      NOP   0;
// CO2D6RV1 PID 001 CO2 D6 RV1
      CALL FC    55 (
           UnitNo                   := #UnitNo,
           PIDRec                   := DB2346.CO2D6RV1,
           SpExt                    := DB2346.DBD  234,
           PVal                     := DB2346.DBD  254,
           OPer                     := PQW  544);

NETWORK
TITLE =unit supply

      UC    FB [#UnitFB];

NETWORK
TITLE =D6_G1  D6_G1
// Act 001
// Box           : VS2-BB
// Output address: Q310.2
      CALL FC    70 (
           UnitNo                   := #UnitNo,
           ActRec                   := DB2340.D6_G1,
           Typ                      := 1,
           FBa                      := #xTmp,
           FBa2                     := I    310.2,
           Out                      := Q    310.2);

NETWORK
TITLE =CO2_D6V2  Ansteuerung D6V2
// Act 002
// Box           : CO2 Dosierung
// Output address: Q61.4
      CALL FC    70 (
           UnitNo                   := #UnitNo,
           ActRec                   := DB2340.CO2_D6V2,
           Typ                      := 0,
           FBa                      := #xTmp,
           FBa2                     := #xTmp,
           Out                      := Q     61.4);

NETWORK
TITLE =CO2_D6V1  Ansteuerung D6V1
// Act 003
// Box           : CO2 Dosierung
// Output address: Q60.4
      CALL FC    70 (
           UnitNo                   := #UnitNo,
           ActRec                   := DB2340.CO2_D6V1,
           Typ                      := 0,
           FBa                      := #xTmp,
           FBa2                     := #xTmp,
           Out                      := Q     60.4);

NETWORK
TITLE =D6RV1  CO2 D6 RV1
// Act 004
// Box           :
// Input address : #xtmp
// Output address: #xtmp
      CALL FC    70 (
           UnitNo                   := #UnitNo,
           ActRec                   := DB2340.D6RV1,
           Typ                      := 4,
           FBa                      := #xTmp,
           FBa2                     := #xTmp,
           Out                      := #xTmp);

END_FUNCTION_BLOCK

FUNCTION_BLOCK FB 1341
TITLE =U034: Well Transfer D6
FAMILY : BOTEC_F1
NAME : UniE
VERSION : 1.2


VAR_TEMP
  CIP : BOOL ;	//CIP active
  UNIM : BOOL ;	//Unit Not In Maintenance
  GenRel : BOOL ;	//general OK (emergency and maintenance OK)
  EStopOK : BOOL ;	//emergency OK
  UnitNo : INT ;	//unit number
  xTmp : BOOL ;	//Temporary Bool
  iTmp : INT ;	//Temporary INT
  rTmp : REAL ;	//Temporary REAL
  dTmp : DINT ;	//Temporary DINT (free for general use)
  RetValInt : INT ;	//return value
END_VAR
BEGIN
NETWORK
TITLE =General

      SET   ;
// Simulation ---------------------------------------------------------------
      A     DB1341.DBX 1357.7;
      CC    FB  1349; // "U034Sim"
      A     DB1341.DBX   17.3;
      =     DB1341.DBX 1357.7; //Help bit for simulation

// get unit number ----------------------------------------------------------
      L     DB1340.DBW    0;
      T     #UnitNo;

// communication ------------------------------------------------------------
      UC    FB  1345; // U034Com

NETWORK
TITLE =Sequence organisation

      CLR   ;
      =     M    122.2;

// sequencer ----------------------------------------------------------------
      A     DB1343.DBX   43.1;
      S     DB1343.DBX   97.3;

      CALL FC    40 (
           UnitNo                   := #UnitNo);

END_FUNCTION_BLOCK

FUNCTION_BLOCK FB 1380
TITLE =U038: Water Treatment 1
FAMILY : BOTEC_F1
NAME : UniA
VERSION : 2.1


VAR_TEMP
  EStopOK : BOOL ;	//auxiliary flag
  CIP : BOOL ;	//CIP Program Selected
  xTmp : BOOL ;	//Temporary Bool(free for general use)
  UnitNo : INT ;	//unit number
  UnitFB : INT ;	//unit expansion FB number
  rTmp : REAL ;	//Temporary REAL (free for general use)
  iTmp : INT ;	//Temporary INT (free for general use)
  dTmp : DINT ;	//Temporary DINT (free for general use)
END_VAR
BEGIN
NETWORK
TITLE =general

      CLR   ;
      =     #xTmp;
      =     #EStopOK;

      L     DB1380.DBW    0;
      T     #UnitNo;
      L     DB1380.DBW    2;
      T     #UnitFB;

NETWORK
TITLE =analog inputs

      NOP   0;
// EW288 AnI 001 Chriwa Filter Durchfluß Produkt
      CALL FC    24 (
           UnitNo                   := #UnitNo,
           AnIRec                   := DB2383.#EW288,
           ValPer                   := 0);//"EW288"

// EW290 AnI 002 Chriwa Filter Durchfluß Spülwasser
      CALL FC    24 (
           UnitNo                   := #UnitNo,
           AnIRec                   := DB2383.#EW290,
           ValPer                   := PIW  290);

// EW284 AnI 003 Chriwa Filter Leitwert
      CALL FC    24 (
           UnitNo                   := #UnitNo,
           AnIRec                   := DB2383.#EW284,
           ValPer                   := PIW  284);

// EW286 AnI 004 Chriwa Filter Trübung
      CALL FC    24 (
           UnitNo                   := #UnitNo,
           AnIRec                   := DB2383.#EW286,
           ValPer                   := PIW  286);

NETWORK
TITLE =Universal value

      NOP   0;
// unv001 UnV 001 Process Status
      CALL FC    27 (
           UnitNo                   := #UnitNo,
           UnVRec                   := DB2385.unv001,
           ValExt                   := DB2385.DBD  234);

// unv002 UnV 002 Universal Value 02
      CALL FC    27 (
           UnitNo                   := #UnitNo,
           UnVRec                   := DB2385.unv002,
           ValExt                   := DB2385.DBD  362);

NETWORK
TITLE =special inputs

      NOP   0;
// CHRIWA_ANF_BRUNNENPUMPE SpI 001 Chriwa Filter
      CALL FC    14 (
           UnitNo                   := #UnitNo,
           SpIRec                   := DB2381.CHRIWA_ANF_BRUNNENPUMPE,
           SpIBit                   := I    280.3);

// CHRIWA_BETRIEB SpI 002 Chriwa Filter
      CALL FC    14 (
           UnitNo                   := #UnitNo,
           SpIRec                   := DB2381.CHRIWA_BETRIEB,
           SpIBit                   := I    280.2);

// CHRIWA_STOERUNG SpI 003 Chriwa Filter
      CALL FC    14 (
           UnitNo                   := #UnitNo,
           SpIRec                   := DB2381.CHRIWA_STOERUNG,
           SpIBit                   := I    280.1);

// CHRIWA_LEBENSBIT SpI 004 Chriwa Filter
      CALL FC    14 (
           UnitNo                   := #UnitNo,
           SpIRec                   := DB2381.CHRIWA_LEBENSBIT,
           SpIBit                   := I    280.0);

// KF1K1 SpI 005 KF1 K1
      CALL FC    14 (
           UnitNo                   := #UnitNo,
           SpIRec                   := DB2381.KF1K1,
           SpIBit                   := #xTmp);

// KF1K2 SpI 006 KF1 K2
      CALL FC    14 (
           UnitNo                   := #UnitNo,
           SpIRec                   := DB2381.KF1K2,
           SpIBit                   := #xTmp);

// KF1_K3 SpI 007 KF1 K3
      CALL FC    14 (
           UnitNo                   := #UnitNo,
           SpIRec                   := DB2381.KF1_K3,
           SpIBit                   := #xTmp);

NETWORK
TITLE =messages

      NOP   0;
// msg001 Msg 001 Message 01
      CALL FC    16 (
           UnitNo                   := #UnitNo,
           MsgRec                   := DB2387.msg001,
           MsgBit                   := DB2387.DBX   82.7);

// msg002 Msg 002 Message 02
      CALL FC    16 (
           UnitNo                   := #UnitNo,
           MsgRec                   := DB2387.msg002,
           MsgBit                   := DB2387.DBX  142.7);

NETWORK
TITLE =unit supply

      UC    FB [#UnitFB];

NETWORK
TITLE =Chriwa_LS_Tank1  Chriwa Filter Tank 1 LS
// Act 005
// Box           : Chriwa
// Output address: Q280.4
      CALL FC    70 (
           UnitNo                   := #UnitNo,
           ActRec                   := DB2380.Chriwa_LS_Tank1,
           Typ                      := 0,
           FBa                      := #xTmp,
           FBa2                     := #xTmp,
           Out                      := Q    280.4);

NETWORK
TITLE =Chriwa_Freigabe_Ruecksp  Chriwa Filter Freigabe zum Rückspülen
// Act 006
// Box           : Chriwa
// Output address: Q280.3
      CALL FC    70 (
           UnitNo                   := #UnitNo,
           ActRec                   := DB2380.Chriwa_Freigabe_Ruecksp,
           Typ                      := 0,
           FBa                      := #xTmp,
           FBa2                     := #xTmp,
           Out                      := Q    280.3);

NETWORK
TITLE =Chriwa_Brunnen_ok  Chriwa Filter Brunnen ok Meldung
// Act 007
// Box           : Chriwa
// Output address: Q280.2
      CALL FC    70 (
           UnitNo                   := #UnitNo,
           ActRec                   := DB2380.Chriwa_Brunnen_ok,
           Typ                      := 0,
           FBa                      := #xTmp,
           FBa2                     := #xTmp,
           Out                      := Q    280.2);

NETWORK
TITLE =Chriwa_Tank_Befuell_Ein  Chriwa Filter Tank Befüllung läuft
// Act 008
// Box           : Chriwa
// Output address: Q280.1
      CALL FC    70 (
           UnitNo                   := #UnitNo,
           ActRec                   := DB2380.Chriwa_Tank_Befuell_Ein,
           Typ                      := 0,
           FBa                      := #xTmp,
           FBa2                     := #xTmp,
           Out                      := Q    280.1);

NETWORK
TITLE =Chriwa_Lebensbit  Chriwa Filter 0,5Hz Lebensbit
// Act 009
// Box           : Chriwa
// Output address: Q280.0
      CALL FC    70 (
           UnitNo                   := #UnitNo,
           ActRec                   := DB2380.Chriwa_Lebensbit,
           Typ                      := 0,
           FBa                      := #xTmp,
           FBa2                     := #xTmp,
           Out                      := Q    280.0);

END_FUNCTION_BLOCK

FUNCTION_BLOCK FB 1381
TITLE =U038: Water Treatment 1
FAMILY : BOTEC_F1
NAME : UniE
VERSION : 1.2


VAR_TEMP
  CIP : BOOL ;	//CIP active
  UNIM : BOOL ;	//Unit Not In Maintenance
  GenRel : BOOL ;	//general OK (emergency and maintenance OK)
  EStopOK : BOOL ;	//emergency OK
  UnitNo : INT ;	//unit number
  xTmp : BOOL ;	//Temporary Bool
  iTmp : INT ;	//Temporary INT
  rTmp : REAL ;	//Temporary REAL
  dTmp : DINT ;	//Temporary DINT (free for general use)
  RetValInt : INT ;	//return value
END_VAR
BEGIN
NETWORK
TITLE =General

      SET   ;
// Simulation ---------------------------------------------------------------
      A     DB1381.DBX 1357.7;
      CC    FB  1389; // "U038Sim"
      A     DB1381.DBX   17.3;
      =     DB1381.DBX 1357.7; //Help bit for simulation

// get unit number ----------------------------------------------------------
      L     DB1380.DBW    0;
      T     #UnitNo;

// CIP ----------------------------------------------------------------------
      L     DB1381.DBD   54;
      L     0;
      <D    ;
      =     #CIP;

// emergency OK -------------------------------------------------------------
      A     DB1385.DBX   27.0; //Emergency Stop OK
      =     #EStopOK;

// Write Unit in Maintenance ------------------------------------------------

      AN    DB1381.DBX   69.7;
      =     #UNIM;

// emergency and maintenance OK ---------------------------------------------
      A     #EStopOK;
      A     #UNIM;
      =     #GenRel;

// communication ------------------------------------------------------------
      UC    FB  1385; // U038Com

NETWORK
TITLE =Analog Inputs

      NOP   0;

// ----------------------------------------------------------
// EW288 Chriwa Filter Durchfluß Produkt
// ----------------------------------------------------------
      L     IW   288;
      ITD   ;
      DTR   ;
      T     DB2383.DBD  214;
      SET   ;
      =     DB2383.DBX  143.5;

      SET   ;
      =     DB2383.DBX  141.5;

// ----------------------------------------------------------
// EW290 Chriwa Filter Durchfluß Spülwasser
// ----------------------------------------------------------
      L     IW   290;
      ITD   ;
      DTR   ;
      T     DB2383.DBD  334;
      SET   ;
      =     DB2383.DBX  263.5;

      SET   ;
      =     DB2383.DBX  261.5;

// ----------------------------------------------------------
// EW284 Chriwa Filter Leitwert
// ----------------------------------------------------------
      L     IW   284;
      ITD   ;
      DTR   ;
      T     DB2383.DBD  454;
      SET   ;
      =     DB2383.DBX  383.5;

      SET   ;
      =     DB2383.DBX  381.5;

// ----------------------------------------------------------
// EW286 Chriwa Filter Trübung
// ----------------------------------------------------------
      L     IW   286;
      ITD   ;
      DTR   ;
      T     DB2383.DBD  574;
      SET   ;
      =     DB2383.DBX  503.5;

      SET   ;
      =     DB2383.DBX  501.5;

NETWORK
TITLE =Universal Value

      NOP   0;

// ----------------------------------------------------------
// unv001 Process Status
// ----------------------------------------------------------
// process value to UnV
//      L     0.000000e+000
//      T     "U038UnVD".unv001.ValExt

// ----------------------------------------------------------
// unv002 Universal Value 02
// ----------------------------------------------------------
// process value to UnV
//      L     0.000000e+000
//      T     "U038UnVD".unv002.ValExt

NETWORK
TITLE =Special Input

      NOP   0;

// ----------------------------------------------------------
// CHRIWA_ANF_BRUNNENPUMPE Chriwa Filter
// ----------------------------------------------------------
      CLR   ;
      =     DB2381.DBX   81.4;
      =     DB2381.DBX   81.5;

// ----------------------------------------------------------
// CHRIWA_BETRIEB Chriwa Filter
// ----------------------------------------------------------
      CLR   ;
      =     DB2381.DBX  141.4;
      =     DB2381.DBX  141.5;

// ----------------------------------------------------------
// CHRIWA_STOERUNG Chriwa Filter
// ----------------------------------------------------------
      SET   ;
      =     DB2381.DBX  201.4;
      CLR   ;
      =     DB2381.DBX  201.5;

// ----------------------------------------------------------
// CHRIWA_LEBENSBIT Chriwa Filter
// ----------------------------------------------------------
      SET   ;
      =     DB2381.DBX  261.4;
      =     DB2381.DBX  261.5;

NETWORK
TITLE =Messages

      NOP   0;

// ----------------------------------------------------------
// msg001 Message 01
// ----------------------------------------------------------
      SET   ;
      R     DB2387.DBX   80.7;
      =     DB2387.DBX   81.4;

      CLR   ;
      =     DB2387.DBX   82.7;

// ----------------------------------------------------------
// msg002 Message 02
// ----------------------------------------------------------
      SET   ;
      R     DB2387.DBX  140.7;
      =     DB2387.DBX  141.4;

      CLR   ;
      =     DB2387.DBX  142.7;

NETWORK
TITLE =Sequence organisation

      CLR   ;
      =     M    122.2;

// SFM supply ----------------------------------------------------------------

// analog value to SFM Chriwa Filter Durchfluß Produkt -----------------------
      L     DB2383.DBD  146;
      T     DB1381.DBD 1122; // !!! insert correct SFM !!!

// analog value to SFM Chriwa Filter Durchfluß Spülwasser -----------------------
      L     DB2383.DBD  266;
      T     DB1381.DBD 1122; // !!! insert correct SFM !!!

// analog value to SFM Chriwa Filter Leitwert -----------------------
      L     DB2383.DBD  386;
      T     DB1381.DBD 1122; // !!! insert correct SFM !!!

// analog value to SFM Chriwa Filter Trübung -----------------------
      L     DB2383.DBD  506;
      T     DB1381.DBD 1122; // !!! insert correct SFM !!!

// Chriwa Status 1
      A     I    292.0; // ERSTFILTRAT
      JC    M100;
      A     I    292.1; // AUS
      JC    M101;
      A     I    292.2; // BEREITSCHAFT
      JC    M102;
      A     I    292.3; // STOP
      JC    M103;
      A     I    292.4; // STÖRUNG
      JC    M104;
      A     I    293.0; // BETRIEB
      JC    M108;
      A     I    293.1; // ENTSPANNE
      JC    M109;
      A     I    293.2; // ABSENKEN
      JC    M110;
      A     I    293.3; // SPÜLEN LUFT
      JC    M111;
      A     I    293.4; // SPÜLEN WASSER/LUFT
      JC    M112;
      A     I    293.5; // FILTERBETTENTL.
      JC    M113;
      A     I    293.6; // SPÜLEN WASSER
      JC    M114;
      A     I    293.7; // AUFFÜLLEN
      JC    M115;
      JU    ELS1;
M100: L     0.000000e+000; // Do 0
      JU    FIN1;
M101: L     1.000000e+000; // Do 1
      JU    FIN1;
M102: L     2.000000e+000; // Do 2
      JU    FIN1;
M103: L     3.000000e+000; // Do 3
      JU    FIN1;
M104: L     4.000000e+000; // Do 4
      JU    FIN1;
M108: L     8.000000e+000; // Do 8
      JU    FIN1;
M109: L     9.000000e+000; // Do 9
      JU    FIN1;
M110: L     1.000000e+001; // Do 10
      JU    FIN1;
M111: L     1.100000e+001; // Do 11
      JU    FIN1;
M112: L     1.200000e+001; // Do 12
      JU    FIN1;
M113: L     1.300000e+001; // Do 13
      JU    FIN1;
M114: L     1.400000e+001; // Do 14
      JU    FIN1;
M115: L     1.500000e+001; // Do 15
      JU    FIN1;
ELS1: L     1.600000e+001; // Do Else
FIN1: T     DB1381.DBD  482;

// Chriwa Status 2
      A     I    294.0; // ERSTFILTRAT
      JC    M200;
      A     I    294.1; // AUS
      JC    M201;
      A     I    294.2; // BEREITSCHAFT
      JC    M202;
      A     I    294.3; // STOP
      JC    M203;
      A     I    294.4; // STÖRUNG
      JC    M204;
      A     I    295.0; // BETRIEB
      JC    M208;
      A     I    295.1; // ENTSPANNE
      JC    M209;
      A     I    295.2; // ABSENKEN
      JC    M210;
      A     I    295.3; // SPÜLEN LUFT
      JC    M211;
      A     I    295.4; // SPÜLEN WASSER/LUFT
      JC    M212;
      A     I    295.5; // FILTERBETTENTL.
      JC    M213;
      A     I    295.6; // SPÜLEN WASSER
      JC    M214;
      A     I    295.7; // AUFFÜLLEN
      JC    M215;
      JU    ELS2;
M200: L     0.000000e+000; // Do 0
      JU    FIN2;
M201: L     1.000000e+000; // Do 1
      JU    FIN2;
M202: L     2.000000e+000; // Do 2
      JU    FIN2;
M203: L     3.000000e+000; // Do 3
      JU    FIN2;
M204: L     4.000000e+000; // Do 4
      JU    FIN2;
M208: L     8.000000e+000; // Do 8
      JU    FIN2;
M209: L     9.000000e+000; // Do 9
      JU    FIN2;
M210: L     1.000000e+001; // Do 10
      JU    FIN2;
M211: L     1.100000e+001; // Do 11
      JU    FIN2;
M212: L     1.200000e+001; // Do 12
      JU    FIN2;
M213: L     1.300000e+001; // Do 13
      JU    FIN2;
M214: L     1.400000e+001; // Do 14
      JU    FIN2;
M215: L     1.500000e+001; // Do 15
      JU    FIN2;
ELS2: L     1.600000e+001; // Do Else
FIN2: T     DB1381.DBD  498;


// sequencer ----------------------------------------------------------------
      A     DB1383.DBX   43.1;
      S     DB1383.DBX   97.3;

      CALL FC    40 (
           UnitNo                   := #UnitNo);

NETWORK
TITLE =Auto / Manual

      SET   ;
      AN    M    122.2;
      JC    MODE;
      AN    M    120.1;

// assign actuator mode
      AN    M    120.1;
      =     DB2380.DBX  105.4;
      =     DB2380.DBX  185.4;
      =     DB2380.DBX  265.4;
      =     DB2380.DBX  425.4;
      =     DB2380.DBX  505.4;
      =     DB2380.DBX  585.4;
      =     DB2380.DBX  665.4;
      =     DB2380.DBX  745.4;



MODE: SET   ;

NETWORK
TITLE =RW5_G1 Gullyventil RW5
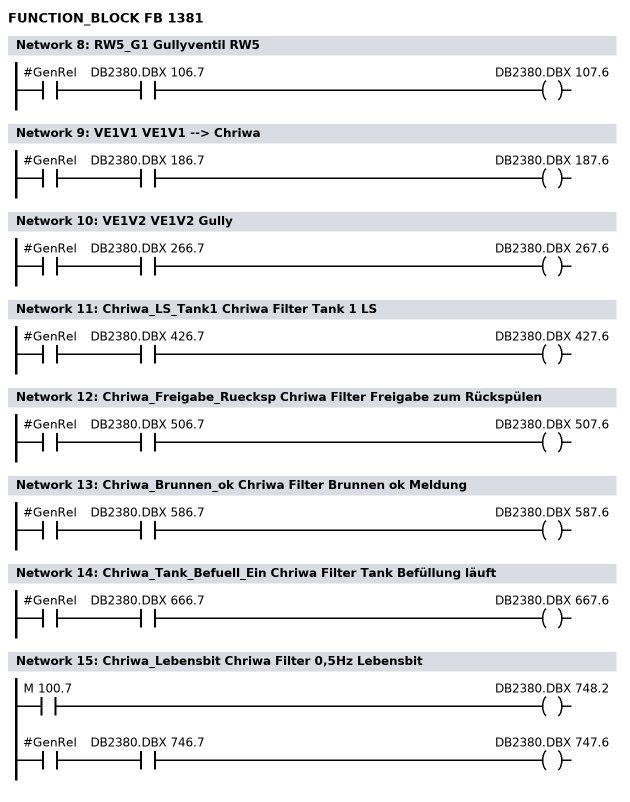

      A     #GenRel;
      A     DB2380.DBX  106.7;
      =     DB2380.DBX  107.6;
NETWORK
TITLE =VE1V1 VE1V1 --> Chriwa

      A     #GenRel;
      A     DB2380.DBX  186.7;
      =     DB2380.DBX  187.6;
NETWORK
TITLE =VE1V2 VE1V2 Gully

      A     #GenRel;
      A     DB2380.DBX  266.7;
      =     DB2380.DBX  267.6;
NETWORK
TITLE =Chriwa_LS_Tank1 Chriwa Filter Tank 1 LS

      A     #GenRel;
      A     DB2380.DBX  426.7;
      =     DB2380.DBX  427.6;
NETWORK
TITLE =Chriwa_Freigabe_Ruecksp Chriwa Filter Freigabe zum Rückspülen

      A     #GenRel;
      A     DB2380.DBX  506.7;
      =     DB2380.DBX  507.6;
NETWORK
TITLE =Chriwa_Brunnen_ok Chriwa Filter Brunnen ok Meldung

      A     #GenRel;
      A     DB2380.DBX  586.7;
      =     DB2380.DBX  587.6;
NETWORK
TITLE =Chriwa_Tank_Befuell_Ein Chriwa Filter Tank Befüllung läuft

      A     #GenRel;
      A     DB2380.DBX  666.7;
      =     DB2380.DBX  667.6;
NETWORK
TITLE =Chriwa_Lebensbit Chriwa Filter 0,5Hz Lebensbit

      A     M    100.7;
      =     DB2380.DBX  748.2;

      A     #GenRel;
      A     DB2380.DBX  746.7;
      =     DB2380.DBX  747.6;
END_FUNCTION_BLOCK

FUNCTION_BLOCK FB 1390
TITLE =U039: Water Treatment 2
FAMILY : BOTEC_F1
NAME : UniA
VERSION : 2.1


VAR_TEMP
  EStopOK : BOOL ;	//auxiliary flag
  CIP : BOOL ;	//CIP Program Selected
  xTmp : BOOL ;	//Temporary Bool(free for general use)
  UnitNo : INT ;	//unit number
  UnitFB : INT ;	//unit expansion FB number
  rTmp : REAL ;	//Temporary REAL (free for general use)
  iTmp : INT ;	//Temporary INT (free for general use)
  dTmp : DINT ;	//Temporary DINT (free for general use)
END_VAR
BEGIN
NETWORK
TITLE =general

      CLR   ;
      =     #xTmp;
      =     #EStopOK;

      L     DB1390.DBW    0;
      T     #UnitNo;
      L     DB1390.DBW    2;
      T     #UnitFB;

NETWORK
TITLE =analog inputs

      NOP   0;
// EW888 AnI 001 Chriwa Filter Durchfluß Produkt
      CALL FC    24 (
           UnitNo                   := #UnitNo,
           AnIRec                   := DB2393.#EW888,
           ValPer                   := IW   888);

// EW890 AnI 002 Chriwa Filter Durchfluß Spülwasser
      CALL FC    24 (
           UnitNo                   := #UnitNo,
           AnIRec                   := DB2393.#EW890,
           ValPer                   := IW   890);

// EW884 AnI 003 Chriwa Filter Leitwert
      CALL FC    24 (
           UnitNo                   := #UnitNo,
           AnIRec                   := DB2393.#EW884,
           ValPer                   := IW   884);

// EW886 AnI 004 Chriwa Filter Trübung
      CALL FC    24 (
           UnitNo                   := #UnitNo,
           AnIRec                   := DB2393.#EW886,
           ValPer                   := IW   886);

NETWORK
TITLE =Universal value

      NOP   0;
// unv001 UnV 001 Process Status
      CALL FC    27 (
           UnitNo                   := #UnitNo,
           UnVRec                   := DB2395.unv001,
           ValExt                   := DB2395.DBD  234);

// unv002 UnV 002 Universal Value 02
      CALL FC    27 (
           UnitNo                   := #UnitNo,
           UnVRec                   := DB2395.unv002,
           ValExt                   := DB2395.DBD  362);

NETWORK
TITLE =special inputs

      NOP   0;
// CHRIWA2_ANF_BRUNNENPUMPE SpI 001 Chriwa Filter
      CALL FC    14 (
           UnitNo                   := #UnitNo,
           SpIRec                   := DB2391.CHRIWA2_ANF_BRUNNENPUMPE,
           SpIBit                   := I    880.3);

// CHRIWA2_BETRIEB SpI 002 Chriwa Filter
      CALL FC    14 (
           UnitNo                   := #UnitNo,
           SpIRec                   := DB2391.CHRIWA2_BETRIEB,
           SpIBit                   := I    880.2);

// CHRIWA2_STOERUNG SpI 003 Chriwa Filter
      CALL FC    14 (
           UnitNo                   := #UnitNo,
           SpIRec                   := DB2391.CHRIWA2_STOERUNG,
           SpIBit                   := I    880.1);

// CHRIWA2_LEBENSBIT SpI 004 Chriwa Filter
      CALL FC    14 (
           UnitNo                   := #UnitNo,
           SpIRec                   := DB2391.CHRIWA2_LEBENSBIT,
           SpIBit                   := I    880.0);

NETWORK
TITLE =messages

      NOP   0;
// msg001 Msg 001 Message 01
      CALL FC    16 (
           UnitNo                   := #UnitNo,
           MsgRec                   := DB2397.msg001,
           MsgBit                   := DB2397.DBX   82.7);

// msg002 Msg 002 Message 02
      CALL FC    16 (
           UnitNo                   := #UnitNo,
           MsgRec                   := DB2397.msg002,
           MsgBit                   := DB2397.DBX  142.7);

NETWORK
TITLE =unit supply

      UC    FB [#UnitFB];

NETWORK
TITLE =Chriwa2_LS_Tank1  Chriwa Filter Tank 1 LS/
// Act 005
// Box           : Chriwa
// Output address: Q880.4
      CALL FC    70 (
           UnitNo                   := #UnitNo,
           ActRec                   := DB2390.Chriwa2_LS_Tank1,
           Typ                      := 0,
           FBa                      := #xTmp,
           FBa2                     := #xTmp,
           Out                      := Q    880.4);

NETWORK
TITLE =Chriwa2_Freigabe_Ruecksp  Chriwa Filter zum Rückspülen
// Act 006
// Box           : Chriwa
// Output address: Q880.3
      CALL FC    70 (
           UnitNo                   := #UnitNo,
           ActRec                   := DB2390.Chriwa2_Freigabe_Ruecksp,
           Typ                      := 0,
           FBa                      := #xTmp,
           FBa2                     := #xTmp,
           Out                      := Q    880.3);

NETWORK
TITLE =Chriwa2_Brunnen_ok  Chriwa Filter Brunnen ok Meldung
// Act 007
// Box           : Chriwa
// Output address: Q880.2
      CALL FC    70 (
           UnitNo                   := #UnitNo,
           ActRec                   := DB2390.Chriwa2_Brunnen_ok,
           Typ                      := 0,
           FBa                      := #xTmp,
           FBa2                     := #xTmp,
           Out                      := Q    880.2);

NETWORK
TITLE =Chriwa2_Tank_Befuell_Ein  Chriwa Filter Tank Befüllung läuft
// Act 008
// Box           : Chriwa
// Output address: Q880.1
      CALL FC    70 (
           UnitNo                   := #UnitNo,
           ActRec                   := DB2390.Chriwa2_Tank_Befuell_Ein,
           Typ                      := 0,
           FBa                      := #xTmp,
           FBa2                     := #xTmp,
           Out                      := Q    880.1);

NETWORK
TITLE =Chriwa2_Lebensbit  Chriwa Filter 0,5Hz Lebensbit
// Act 009
// Box           : Chriwa
// Output address: Q880.0
      CALL FC    70 (
           UnitNo                   := #UnitNo,
           ActRec                   := DB2390.Chriwa2_Lebensbit,
           Typ                      := 0,
           FBa                      := #xTmp,
           FBa2                     := #xTmp,
           Out                      := Q    880.0);

END_FUNCTION_BLOCK

FUNCTION_BLOCK FB 1391
TITLE =U039: Water Treatment 2
FAMILY : BOTEC_F1
NAME : UniE
VERSION : 1.2


VAR_TEMP
  CIP : BOOL ;	//CIP active
  UNIM : BOOL ;	//Unit Not In Maintenance
  GenRel : BOOL ;	//general OK (emergency and maintenance OK)
  EStopOK : BOOL ;	//emergency OK
  UnitNo : INT ;	//unit number
  xTmp : BOOL ;	//Temporary Bool
  iTmp : INT ;	//Temporary INT
  rTmp : REAL ;	//Temporary REAL
  dTmp : DINT ;	//Temporary DINT (free for general use)
  RetValInt : INT ;	//return value
END_VAR
BEGIN
NETWORK
TITLE =General

      SET   ;
// Simulation ---------------------------------------------------------------
      A     DB1391.DBX 1357.7;
      CC    FB  1399; // "U039Sim"
      A     DB1391.DBX   17.3;
      =     DB1391.DBX 1357.7; //Help bit for simulation

// get unit number ----------------------------------------------------------
      L     DB1390.DBW    0;
      T     #UnitNo;

// CIP ----------------------------------------------------------------------
      L     DB1391.DBD   54;
      L     0;
      <D    ;
      =     #CIP;

// emergency OK -------------------------------------------------------------
      A     DB1395.DBX   27.0; //Emergency Stop OK
      =     #EStopOK;

// Write Unit in Maintenance ------------------------------------------------

      AN    DB1391.DBX   69.7;
      =     #UNIM;

// emergency and maintenance OK ---------------------------------------------
      A     #EStopOK;
      A     #UNIM;
      =     #GenRel;

// communication ------------------------------------------------------------
      UC    FB  1395; // U039Com

NETWORK
TITLE =Analog Inputs

      NOP   0;

// ----------------------------------------------------------
// EW888 Chriwa Filter Durchfluß Produkt
// ----------------------------------------------------------
      L     IW   888;
      ITD   ;
      DTR   ;
      T     DB2393.DBD  214;
      SET   ;
      =     DB2393.DBX  143.5;


      L     DB1391.DBD 1118; // !!! insert correct SFM !!!
      T     DB2393.DBD  238;

      SET   ;
      =     DB2393.DBX  141.5;

// ----------------------------------------------------------
// EW890 Chriwa Filter Durchfluß Spülwasser
// ----------------------------------------------------------
      L     IW   890;
      ITD   ;
      DTR   ;
      T     DB2393.DBD  334;
      SET   ;
      =     DB2393.DBX  263.5;

      L     DB1391.DBD 1118; // !!! insert correct SFM !!!
      T     DB2393.DBD  358;

      SET   ;
      =     DB2393.DBX  261.5;

// ----------------------------------------------------------
// EW884 Chriwa Filter Leitwert
// ----------------------------------------------------------
      L     IW   884;
      ITD   ;
      DTR   ;
      T     DB2393.DBD  454;
      SET   ;
      =     DB2393.DBX  383.5;

      L     DB1391.DBD 1118; // !!! insert correct SFM !!!
      T     DB2393.DBD  478;

      SET   ;
      =     DB2393.DBX  381.5;

// ----------------------------------------------------------
// EW886 Chriwa Filter Trübung
// ----------------------------------------------------------
      L     IW   886;
      ITD   ;
      DTR   ;
      T     DB2393.DBD  574;
      SET   ;
      =     DB2393.DBX  503.5;

      L     DB1391.DBD 1118; // !!! insert correct SFM !!!
      T     DB2393.DBD  598;

      SET   ;
      =     DB2393.DBX  501.5;

NETWORK
TITLE =Universal Value

      NOP   0;

// ----------------------------------------------------------
// unv001 Process Status
// ----------------------------------------------------------
// process value to UnV
//      L     0.000000e+000
//      T     "U039UnVD".unv001.ValExt

// ----------------------------------------------------------
// unv002 Universal Value 02
// ----------------------------------------------------------
// process value to UnV
//      L     0.000000e+000
//      T     "U039UnVD".unv002.ValExt

NETWORK
TITLE =Special Input

      NOP   0;

// ----------------------------------------------------------
// CHRIWA2_ANF_BRUNNENPUMPE Chriwa Filter
// ----------------------------------------------------------
      CLR   ;
      =     DB2391.DBX   81.4;
      =     DB2391.DBX   81.5;

// ----------------------------------------------------------
// CHRIWA2_BETRIEB Chriwa Filter
// ----------------------------------------------------------
      CLR   ;
      =     DB2391.DBX  141.4;
      =     DB2391.DBX  141.5;

// ----------------------------------------------------------
// CHRIWA2_STOERUNG Chriwa Filter
// ----------------------------------------------------------
      SET   ;
      =     DB2391.DBX  201.4;
      CLR   ;
      =     DB2391.DBX  201.5;

// ----------------------------------------------------------
// CHRIWA2_LEBENSBIT Chriwa Filter
// ----------------------------------------------------------
      SET   ;
      =     DB2391.DBX  261.4;
      =     DB2391.DBX  261.5;

NETWORK
TITLE =Messages

      NOP   0;

// ----------------------------------------------------------
// msg001 Message 01
// ----------------------------------------------------------
      SET   ;
      R     DB2397.DBX   80.7;
      =     DB2397.DBX   81.4;

      CLR   ;
      =     DB2397.DBX   82.7;

// ----------------------------------------------------------
// msg002 Message 02
// ----------------------------------------------------------
      SET   ;
      R     DB2397.DBX  140.7;
      =     DB2397.DBX  141.4;

      CLR   ;
      =     DB2397.DBX  142.7;

NETWORK
TITLE =Sequence organisation

      CLR   ;
      =     M    122.2;

// SFM supply ----------------------------------------------------------------

// analog value to SFM Chriwa Filter Durchfluß Produkt -----------------------
      L     DB2393.DBD  146;
      T     DB1391.DBD 1122; // !!! insert correct SFM !!!

// analog value to SFM Chriwa Filter Durchfluß Spülwasser -----------------------
      L     DB2393.DBD  266;
      T     DB1391.DBD 1122; // !!! insert correct SFM !!!

// analog value to SFM Chriwa Filter Leitwert -----------------------
      L     DB2393.DBD  386;
      T     DB1391.DBD 1122; // !!! insert correct SFM !!!

// analog value to SFM Chriwa Filter Trübung -----------------------
      L     DB2393.DBD  506;
      T     DB1391.DBD 1122; // !!! insert correct SFM !!!


// Chriwa Status 1
      A     I    892.0; // ERSTFILTRAT
      JC    M100;
      A     I    892.1; // AUS
      JC    M101;
      A     I    892.2; // BEREITSCHAFT
      JC    M102;
      A     I    892.3; // STOP
      JC    M103;
      A     I    892.4; // STÖRUNG
      JC    M104;
      A     I    893.0; // BETRIEB
      JC    M108;
      A     I    893.1; // ENTSPANNE
      JC    M109;
      A     I    893.2; // ABSENKEN
      JC    M110;
      A     I    893.3; // SPÜLEN LUFT
      JC    M111;
      A     I    893.4; // SPÜLEN WASSER/LUFT
      JC    M112;
      A     I    893.5; // FILTERBETTENTL.
      JC    M113;
      A     I    893.6; // SPÜLEN WASSER
      JC    M114;
      A     I    893.7; // AUFFÜLLEN
      JC    M115;
      JU    ELS1;
M100: L     0.000000e+000; // Do 0
      JU    FIN1;
M101: L     1.000000e+000; // Do 1
      JU    FIN1;
M102: L     2.000000e+000; // Do 2
      JU    FIN1;
M103: L     3.000000e+000; // Do 3
      JU    FIN1;
M104: L     4.000000e+000; // Do 4
      JU    FIN1;
M108: L     8.000000e+000; // Do 8
      JU    FIN1;
M109: L     9.000000e+000; // Do 9
      JU    FIN1;
M110: L     1.000000e+001; // Do 10
      JU    FIN1;
M111: L     1.100000e+001; // Do 11
      JU    FIN1;
M112: L     1.200000e+001; // Do 12
      JU    FIN1;
M113: L     1.300000e+001; // Do 13
      JU    FIN1;
M114: L     1.400000e+001; // Do 14
      JU    FIN1;
M115: L     1.500000e+001; // Do 15
      JU    FIN1;
ELS1: L     1.600000e+001; // Do Else
FIN1: T     DB1391.DBD  482;

// Chriwa Status 2
      A     I    894.0; // ERSTFILTRAT
      JC    M200;
      A     I    894.1; // AUS
      JC    M201;
      A     I    894.2; // BEREITSCHAFT
      JC    M202;
      A     I    894.3; // STOP
      JC    M203;
      A     I    894.4; // STÖRUNG
      JC    M204;
      A     I    895.0; // BETRIEB
      JC    M208;
      A     I    895.1; // ENTSPANNE
      JC    M209;
      A     I    895.2; // ABSENKEN
      JC    M210;
      A     I    895.3; // SPÜLEN LUFT
      JC    M211;
      A     I    895.4; // SPÜLEN WASSER/LUFT
      JC    M212;
      A     I    895.5; // FILTERBETTENTL.
      JC    M213;
      A     I    895.6; // SPÜLEN WASSER
      JC    M214;
      A     I    895.7; // AUFFÜLLEN
      JC    M215;
      JU    ELS2;
M200: L     0.000000e+000; // Do 0
      JU    FIN2;
M201: L     1.000000e+000; // Do 1
      JU    FIN2;
M202: L     2.000000e+000; // Do 2
      JU    FIN2;
M203: L     3.000000e+000; // Do 3
      JU    FIN2;
M204: L     4.000000e+000; // Do 4
      JU    FIN2;
M208: L     8.000000e+000; // Do 8
      JU    FIN2;
M209: L     9.000000e+000; // Do 9
      JU    FIN2;
M210: L     1.000000e+001; // Do 10
      JU    FIN2;
M211: L     1.100000e+001; // Do 11
      JU    FIN2;
M212: L     1.200000e+001; // Do 12
      JU    FIN2;
M213: L     1.300000e+001; // Do 13
      JU    FIN2;
M214: L     1.400000e+001; // Do 14
      JU    FIN2;
M215: L     1.500000e+001; // Do 15
      JU    FIN2;
ELS2: L     1.600000e+001; // Do Else
FIN2: T     DB1391.DBD  498;


// sequencer ----------------------------------------------------------------
      A     DB1393.DBX   43.1;
      S     DB1393.DBX   97.3;

      CALL FC    40 (
           UnitNo                   := #UnitNo);

NETWORK
TITLE =Auto / Manual

      SET   ;
      AN    M    122.2;
      JC    MODE;
      AN    M    120.1;

// assign actuator mode
      AN    M    120.1;
      =     DB2390.DBX  105.4;
      =     DB2390.DBX  185.4;
      =     DB2390.DBX  265.4;
      =     DB2390.DBX  425.4;
      =     DB2390.DBX  505.4;
      =     DB2390.DBX  585.4;
      =     DB2390.DBX  665.4;
      =     DB2390.DBX  745.4;



MODE: SET   ;

NETWORK
TITLE =RW6_G1 Gullyventil RW6
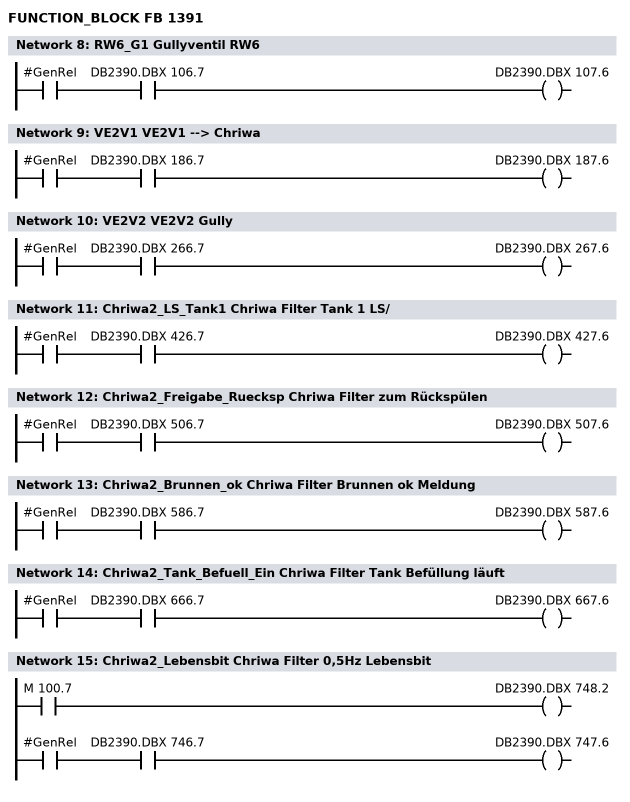

      A     #GenRel;
      A     DB2390.DBX  106.7;
      =     DB2390.DBX  107.6;
NETWORK
TITLE =VE2V1 VE2V1 --> Chriwa

      A     #GenRel;
      A     DB2390.DBX  186.7;
      =     DB2390.DBX  187.6;
NETWORK
TITLE =VE2V2 VE2V2 Gully

      A     #GenRel;
      A     DB2390.DBX  266.7;
      =     DB2390.DBX  267.6;
NETWORK
TITLE =Chriwa2_LS_Tank1 Chriwa Filter Tank 1 LS/

      A     #GenRel;
      A     DB2390.DBX  426.7;
      =     DB2390.DBX  427.6;
NETWORK
TITLE =Chriwa2_Freigabe_Ruecksp Chriwa Filter zum Rückspülen

      A     #GenRel;
      A     DB2390.DBX  506.7;
      =     DB2390.DBX  507.6;
NETWORK
TITLE =Chriwa2_Brunnen_ok Chriwa Filter Brunnen ok Meldung

      A     #GenRel;
      A     DB2390.DBX  586.7;
      =     DB2390.DBX  587.6;
NETWORK
TITLE =Chriwa2_Tank_Befuell_Ein Chriwa Filter Tank Befüllung läuft

      A     #GenRel;
      A     DB2390.DBX  666.7;
      =     DB2390.DBX  667.6;
NETWORK
TITLE =Chriwa2_Lebensbit Chriwa Filter 0,5Hz Lebensbit

      A     M    100.7;
      =     DB2390.DBX  748.2;

      A     #GenRel;
      A     DB2390.DBX  746.7;
      =     DB2390.DBX  747.6;
END_FUNCTION_BLOCK

FUNCTION_BLOCK FB 1400
TITLE =U040: Water Treatment General
FAMILY : BOTEC_F1
NAME : UniA
VERSION : 2.1


VAR_TEMP
  EStopOK : BOOL ;	//auxiliary flag
  CIP : BOOL ;	//CIP Program Selected
  xTmp : BOOL ;	//Temporary Bool(free for general use)
  UnitNo : INT ;	//unit number
  UnitFB : INT ;	//unit expansion FB number
  rTmp : REAL ;	//Temporary REAL (free for general use)
  iTmp : INT ;	//Temporary INT (free for general use)
  dTmp : DINT ;	//Temporary DINT (free for general use)
END_VAR
BEGIN
NETWORK
TITLE =general

      CLR   ;
      =     #xTmp;
      =     #EStopOK;

      L     DB1400.DBW    0;
      T     #UnitNo;
      L     DB1400.DBW    2;
      T     #UnitFB;

NETWORK
TITLE =Universal value

      NOP   0;
// unv001 UnV 001 Process Status
      CALL FC    27 (
           UnitNo                   := #UnitNo,
           UnVRec                   := DB2405.unv001,
           ValExt                   := DB2405.DBD  234);

// unv002 UnV 002 Universal Value 02
      CALL FC    27 (
           UnitNo                   := #UnitNo,
           UnVRec                   := DB2405.unv002,
           ValExt                   := DB2405.DBD  362);

NETWORK
TITLE =special inputs

      NOP   0;
// RM_VEE_P1 SpI 001 UEBERGABEKONTAKTE VON LT
      CALL FC    14 (
           UnitNo                   := #UnitNo,
           SpIRec                   := DB2401.RM_VEE_P1,
           SpIBit                   := I    108.3);

// RM_VEE_P2 SpI 002 UEBERGABEKONTAKTE VON LT
      CALL FC    14 (
           UnitNo                   := #UnitNo,
           SpIRec                   := DB2401.RM_VEE_P2,
           SpIBit                   := I    108.4);

// BETR_BRUNNEN_7 SpI 003 MELDUNG VON VEE
      CALL FC    14 (
           UnitNo                   := #UnitNo,
           SpIRec                   := DB2401.BETR_BRUNNEN_7,
           SpIBit                   := I     14.0);

// BETR_BRUNNEN_2B SpI 004 MELDUNG VON VEE
      CALL FC    14 (
           UnitNo                   := #UnitNo,
           SpIRec                   := DB2401.BETR_BRUNNEN_2B,
           SpIBit                   := I     14.1);

// BETR_BRUNNEN_3 SpI 005 MELDUNG VON VEE
      CALL FC    14 (
           UnitNo                   := #UnitNo,
           SpIRec                   := DB2401.BETR_BRUNNEN_3,
           SpIBit                   := I     14.2);

// BETR_BRUNNEN_2A SpI 006 MELDUNG VON VEE
      CALL FC    14 (
           UnitNo                   := #UnitNo,
           SpIRec                   := DB2401.BETR_BRUNNEN_2A,
           SpIBit                   := I     14.3);

NETWORK
TITLE =messages

      NOP   0;
// msg001 Msg 001 Message 01
      CALL FC    16 (
           UnitNo                   := #UnitNo,
           MsgRec                   := DB2407.msg001,
           MsgBit                   := DB2407.DBX   82.7);

// msg002 Msg 002 Message 02
      CALL FC    16 (
           UnitNo                   := #UnitNo,
           MsgRec                   := DB2407.msg002,
           MsgBit                   := DB2407.DBX  142.7);

NETWORK
TITLE =unit supply

      UC    FB [#UnitFB];
END_FUNCTION_BLOCK

FUNCTION_BLOCK FB 1401
TITLE =U040: Water Treatment General
FAMILY : BOTEC_F1
NAME : UniE
VERSION : 1.2


VAR_TEMP
  CIP : BOOL ;	//CIP active
  UNIM : BOOL ;	//Unit Not In Maintenance
  GenRel : BOOL ;	//general OK (emergency and maintenance OK)
  EStopOK : BOOL ;	//emergency OK
  UnitNo : INT ;	//unit number
  xTmp : BOOL ;	//Temporary Bool
  iTmp : INT ;	//Temporary INT
  rTmp : REAL ;	//Temporary REAL
  dTmp : DINT ;	//Temporary DINT (free for general use)
  RetValInt : INT ;	//return value
END_VAR
BEGIN
NETWORK
TITLE =General

      SET   ;
// Simulation ---------------------------------------------------------------
      A     DB1401.DBX 1357.7;
      CC    FB  1409; // "U040Sim"
      A     DB1401.DBX   17.3;
      =     DB1401.DBX 1357.7; //Help bit for simulation

// get unit number ----------------------------------------------------------
      L     DB1400.DBW    0;
      T     #UnitNo;

// CIP ----------------------------------------------------------------------
      L     DB1401.DBD   54;
      L     0;
      <D    ;
      =     #CIP;

// emergency OK -------------------------------------------------------------
      A     DB1405.DBX   27.0; //Emergency Stop OK
      =     #EStopOK;

// Write Unit in Maintenance ------------------------------------------------

      AN    DB1401.DBX   69.7;
      =     #UNIM;

// emergency and maintenance OK ---------------------------------------------
      A     #EStopOK;
      A     #UNIM;
      =     #GenRel;

// communication ------------------------------------------------------------
      UC    FB  1405; // U040Com

NETWORK
TITLE =Universal Value

      NOP   0;

// ----------------------------------------------------------
// unv001 Process Status
// ----------------------------------------------------------
// process value to UnV
//      L     0.000000e+000
//      T     "U040UnVD".unv001.ValExt

// ----------------------------------------------------------
// unv002 Universal Value 02
// ----------------------------------------------------------
// process value to UnV
//      L     0.000000e+000
//      T     "U040UnVD".unv002.ValExt

NETWORK
TITLE =Special Input

      NOP   0;

// ----------------------------------------------------------
// RM_VEE_P1 UEBERGABEKONTAKTE VON LT
// ----------------------------------------------------------
      SET   ;
      =     DB2401.DBX   81.4;
      =     DB2401.DBX   81.5;

// ----------------------------------------------------------
// RM_VEE_P2 UEBERGABEKONTAKTE VON LT
// ----------------------------------------------------------
      SET   ;
      =     DB2401.DBX  141.4;
      =     DB2401.DBX  141.5;

// ----------------------------------------------------------
// BETR_BRUNNEN_7 MELDUNG VON VEE
// ----------------------------------------------------------
      SET   ;
      =     DB2401.DBX  201.4;
      =     DB2401.DBX  201.5;

// ----------------------------------------------------------
// BETR_BRUNNEN_2B MELDUNG VON VEE
// ----------------------------------------------------------
      SET   ;
      =     DB2401.DBX  261.4;
      =     DB2401.DBX  261.5;

// ----------------------------------------------------------
// BETR_BRUNNEN_3 MELDUNG VON VEE
// ----------------------------------------------------------
      SET   ;
      =     DB2401.DBX  321.4;
      =     DB2401.DBX  321.5;

// ----------------------------------------------------------
// BETR_BRUNNEN_2A MELDUNG VON VEE
// ----------------------------------------------------------
      SET   ;
      =     DB2401.DBX  381.4;
      =     DB2401.DBX  381.5;

NETWORK
TITLE =Messages

      NOP   0;

// ----------------------------------------------------------
// msg001 Message 01
// ----------------------------------------------------------
      SET   ;
      R     DB2407.DBX   80.7;
      =     DB2407.DBX   81.4;

      CLR   ;
      =     DB2407.DBX   82.7;

// ----------------------------------------------------------
// msg002 Message 02
// ----------------------------------------------------------
      SET   ;
      R     DB2407.DBX  140.7;
      =     DB2407.DBX  141.4;

      CLR   ;
      =     DB2407.DBX  142.7;

NETWORK
TITLE =Sequence organisation

      CLR   ;
      =     M    122.2;

// SFM supply ----------------------------------------------------------------

// sequencer ----------------------------------------------------------------
      A     DB1403.DBX   43.1;
      S     DB1403.DBX   97.3;

      CALL FC    40 (
           UnitNo                   := #UnitNo);

NETWORK
TITLE =Auto / Manual

      SET   ;
      AN    M    122.2;
      JC    MODE;
      AN    M    120.1;




MODE: SET   ;

END_FUNCTION_BLOCK

FUNCTION_BLOCK FB 1430
TITLE =U043: Water Transfer Plant 3
FAMILY : BOTEC_F1
NAME : UniA
VERSION : 2.1


VAR_TEMP
  EStopOK : BOOL ;	//auxiliary flag
  CIP : BOOL ;	//CIP Program Selected
  xTmp : BOOL ;	//Temporary Bool(free for general use)
  UnitNo : INT ;	//unit number
  UnitFB : INT ;	//unit expansion FB number
  rTmp : REAL ;	//Temporary REAL (free for general use)
  iTmp : INT ;	//Temporary INT (free for general use)
  dTmp : DINT ;	//Temporary DINT (free for general use)
END_VAR
BEGIN
NETWORK
TITLE =general

      CLR   ;
      =     #xTmp;
      =     #EStopOK;

      L     DB1430.DBW    0;
      T     #UnitNo;
      L     DB1430.DBW    2;
      T     #UnitFB;

NETWORK
TITLE =Universal value

      NOP   0;
// unv001 UnV 001 Process Status
      CALL FC    27 (
           UnitNo                   := #UnitNo,
           UnVRec                   := DB2435.unv001,
           ValExt                   := DB2435.DBD  234);

// unv002 UnV 002 Universal Value 02
      CALL FC    27 (
           UnitNo                   := #UnitNo,
           UnVRec                   := DB2435.unv002,
           ValExt                   := DB2435.DBD  362);

// unv003 UnV 003 Universal Value 03
      CALL FC    27 (
           UnitNo                   := #UnitNo,
           UnVRec                   := DB2435.unv003,
           ValExt                   := DB2435.DBD  490);

// unv004 UnV 004 Universal Value 04
      CALL FC    27 (
           UnitNo                   := #UnitNo,
           UnVRec                   := DB2435.unv004,
           ValExt                   := DB2435.DBD  618);

NETWORK
TITLE =special inputs

      NOP   0;
// RM_KEG_V14 SpI 001 KEG_V14
      CALL FC    14 (
           UnitNo                   := #UnitNo,
           SpIRec                   := DB2431.RM_KEG_V14,
           SpIBit                   := I     33.1);

NETWORK
TITLE =messages

      NOP   0;
// msg001 Msg 001 Message 01
      CALL FC    16 (
           UnitNo                   := #UnitNo,
           MsgRec                   := DB2437.msg001,
           MsgBit                   := DB2437.DBX   82.7);

// msg002 Msg 002 Message 02
      CALL FC    16 (
           UnitNo                   := #UnitNo,
           MsgRec                   := DB2437.msg002,
           MsgBit                   := DB2437.DBX  142.7);

// msg003 Msg 003 Message 03
      CALL FC    16 (
           UnitNo                   := #UnitNo,
           MsgRec                   := DB2437.msg003,
           MsgBit                   := DB2437.DBX  202.7);

NETWORK
TITLE =unit supply

      UC    FB [#UnitFB];

NETWORK
TITLE =KEG_RWP  KEG Reinwasserpumpe Freigabe (dummy)
// Act 001
// Box           : S6 U6.3
// Input address : I6.5
// Output address: Q6.5
      CALL FC    70 (
           UnitNo                   := #UnitNo,
           ActRec                   := DB2430.Act1,
           Typ                      := 0,//3 (RM wechselt nicht)
           FBa                      := #xTmp,
           FBa2                     := I      6.5,
           Out                      := Q      6.5);

NETWORK
TITLE =KEG_V11  KEG_V11
// Act 002
// Box           : VS-KEG
// Input address : I32.6
// Output address: Q32.6
      CALL FC    70 (
           UnitNo                   := #UnitNo,
           ActRec                   := DB2430.KEG_V11,
           Typ                      := 1,
           FBa                      := #xTmp,
           FBa2                     := I     32.6,
           Out                      := Q     32.6);

NETWORK
TITLE =KEG_V12  KEG_V12
// Act 003
// Box           : VS-KEG
// Input address : I32.7
// Output address: Q32.7
      CALL FC    70 (
           UnitNo                   := #UnitNo,
           ActRec                   := DB2430.KEG_V12,
           Typ                      := 1,
           FBa                      := #xTmp,
           FBa2                     := I     32.7,
           Out                      := Q     32.7);

NETWORK
TITLE =KEG_V13  KEG_V13
// Act 004
// Box           : VS-KEG
// Input address : I33.0
// Output address: Q33.0
      CALL FC    70 (
           UnitNo                   := #UnitNo,
           ActRec                   := DB2430.KEG_V13,
           Typ                      := 1,
           FBa                      := #xTmp,
           FBa2                     := I     33.0,
           Out                      := Q     33.0);

NETWORK
TITLE =KEG_RV2
// Act 006
// Box           : Ventilinsel 5
// Input address : I339.7
// Output address: Q339.7
      CALL FC    70 (
           UnitNo                   := #UnitNo,
           ActRec                   := DB2430.KEG_RV2,
           Typ                      := 1,
           FBa                      := #xTmp,
           FBa2                     := I    339.7,
           Out                      := Q    339.7);

NETWORK
TITLE =U43_Act010
// Act 010
// Box           :
// Output address: #DummyBool
      CALL FC    70 (
           UnitNo                   := #UnitNo,
           ActRec                   := DB2430.U43_Act010,
           Typ                      := 0,
           FBa                      := #xTmp,
           FBa2                     := #xTmp,
           Out                      := #xTmp);

END_FUNCTION_BLOCK

FUNCTION_BLOCK FB 1431
TITLE =U043: Water Transfer Plant 3
FAMILY : BOTEC_F1
NAME : UniE
VERSION : 1.2


VAR_TEMP
  CIP : BOOL ;	//CIP active
  UNIM : BOOL ;	//Unit Not In Maintenance
  GenRel : BOOL ;	//general OK (emergency and maintenance OK)
  EStopOK : BOOL ;	//emergency OK
  UnitNo : INT ;	//unit number
  xTmp : BOOL ;	//Temporary Bool
  iTmp : INT ;	//Temporary INT
  rTmp : REAL ;	//Temporary REAL
  dTmp : DINT ;	//Temporary DINT (free for general use)
  RetValInt : INT ;	//return value
END_VAR
BEGIN
NETWORK
TITLE =General

      SET   ;
// Simulation ---------------------------------------------------------------
      A     DB1431.DBX 1357.7;
      CC    FB  1439; // "U043Sim"
      A     DB1431.DBX   17.3;
      =     DB1431.DBX 1357.7; //Help bit for simulation

// get unit number ----------------------------------------------------------
      L     DB1430.DBW    0;
      T     #UnitNo;

// communication ------------------------------------------------------------
      UC    FB  1435;

NETWORK
TITLE =Sequence organisation

      CLR   ;
      =     M    122.2;

// CIP Counter
      CALL FC    29 (
           UnitNo                   := #UnitNo,
           Value                    := DB1435.DBD   54,
           Enable                   := TRUE,
           Down                     := FALSE,
           OriginDetect             := 0.000000e+000,
           MaxDiffPS                := 1.000000e+000,
           SFMRec                   := DB1431.Seq.SFM[15],
           ValueOld                 := DB1431.DBD 1418);

// CIP Counter
      CALL FC    29 (
           UnitNo                   := #UnitNo,
           Value                    := DB1435.DBD   54,
           Enable                   := TRUE,
           Down                     := FALSE,
           OriginDetect             := 0.000000e+000,
           MaxDiffPS                := 1.000000e+000,
           SFMRec                   := DB1431.Seq.SFM[15],
           ValueOld                 := DB1431.DBD 1418);

// sequencer ----------------------------------------------------------------
      A     DB1433.DBX   43.1;
      S     DB1433.DBX   97.3;

      CALL FC    40 (
           UnitNo                   := #UnitNo);

END_FUNCTION_BLOCK

FUNCTION_BLOCK FB 1450
TITLE =U045: Water Transfer Plant 5
FAMILY : BOTEC_F1
NAME : UniA
VERSION : 2.1


VAR_TEMP
  EStopOK : BOOL ;	//auxiliary flag
  CIP : BOOL ;	//CIP Program Selected
  xTmp : BOOL ;	//Temporary Bool(free for general use)
  UnitNo : INT ;	//unit number
  UnitFB : INT ;	//unit expansion FB number
  rTmp : REAL ;	//Temporary REAL (free for general use)
  iTmp : INT ;	//Temporary INT (free for general use)
  dTmp : DINT ;	//Temporary DINT (free for general use)
END_VAR
BEGIN
NETWORK
TITLE =general

      CLR   ;
      =     #xTmp;
      =     #EStopOK;

      L     DB1450.DBW    0;
      T     #UnitNo;
      L     DB1450.DBW    2;
      T     #UnitFB;

NETWORK
TITLE =Universal value

      NOP   0;
// unv001 UnV 001 Process Status
      CALL FC    27 (
           UnitNo                   := #UnitNo,
           UnVRec                   := DB2455.unv001,
           ValExt                   := DB2455.DBD  234);

// unv002 UnV 002 Universal Value 02
      CALL FC    27 (
           UnitNo                   := #UnitNo,
           UnVRec                   := DB2455.unv002,
           ValExt                   := DB2455.DBD  362);

// unv003 UnV 003 Universal Value 03
      CALL FC    27 (
           UnitNo                   := #UnitNo,
           UnVRec                   := DB2455.unv003,
           ValExt                   := DB2455.DBD  490);

// unv004 UnV 004 Universal Value 04
      CALL FC    27 (
           UnitNo                   := #UnitNo,
           UnVRec                   := DB2455.unv004,
           ValExt                   := DB2455.DBD  618);

NETWORK
TITLE =special inputs

      NOP   0;
// U45_SpI001 SpI 001 spare
//      CALL  "SI1"
//       UnitNo:=#UnitNo
//       SpIRec:="U045SpID".U45_SpI001
//       SpIBit:=#xTmp

NETWORK
TITLE =messages

      NOP   0;
// msg001 Msg 001 Message 01
      CALL FC    16 (
           UnitNo                   := #UnitNo,
           MsgRec                   := DB2457.msg001,
           MsgBit                   := DB2457.DBX   82.7);

// msg002 Msg 002 Message 02
      CALL FC    16 (
           UnitNo                   := #UnitNo,
           MsgRec                   := DB2457.msg002,
           MsgBit                   := DB2457.DBX  142.7);

// msg003 Msg 003 Message 03
      CALL FC    16 (
           UnitNo                   := #UnitNo,
           MsgRec                   := DB2457.msg003,
           MsgBit                   := DB2457.DBX  202.7);

NETWORK
TITLE =unit supply

      UC    FB [#UnitFB];

NETWORK
TITLE =Act1  Wasserpumpe
// Act 001
// Box           :
// Input address : #xTmp
// Output address: #xTmp
      CALL FC    70 (
           UnitNo                   := #UnitNo,
           ActRec                   := DB2450.Act1,
           Typ                      := 0,
           FBa                      := I    199.1,
           FBa2                     := #xTmp,
           Out                      := Q    199.1);

NETWORK
TITLE =A5_V11  Filter A5 V11
// Act 002
// Box           : VSA5
// Input address : I192.6
// Output address: Q192.6
      CALL FC    70 (
           UnitNo                   := #UnitNo,
           ActRec                   := DB2450.A5_V11,
           Typ                      := 1,
           FBa                      := #xTmp,
           FBa2                     := I    192.6,
           Out                      := Q    192.6);

NETWORK
TITLE =A5_V12  Filter A5 V12
// Act 003
// Box           : VSA5
// Input address : I192.7
// Output address: Q192.7
      CALL FC    70 (
           UnitNo                   := #UnitNo,
           ActRec                   := DB2450.A5_V12,
           Typ                      := 1,
           FBa                      := #xTmp,
           FBa2                     := I    192.7,
           Out                      := Q    192.7);

NETWORK
TITLE =A5_V13  Filter A5 V13
// Act 004
// Box           : VSA5
// Input address : I193.0
// Output address: Q193.0
      CALL FC    70 (
           UnitNo                   := #UnitNo,
           ActRec                   := DB2450.A5_V13,
           Typ                      := 1,
           FBa                      := #xTmp,
           FBa2                     := I    193.0,
           Out                      := Q    193.0);

NETWORK
TITLE =RV1_A5
// Act 005
// Box           : Ventilinsel 3
// Input address : I327.5
// Output address: Q327.5
      CALL FC    70 (
           UnitNo                   := #UnitNo,
           ActRec                   := DB2450.RV1_A5,
           Typ                      := 1,
           FBa                      := #xTmp,
           FBa2                     := I    327.5,
           Out                      := Q    327.5);

NETWORK
TITLE =RV2_A5
// Act 006
// Box           : Ventilinsel 3
// Input address : I327.6
// Output address: Q327.6
      CALL FC    70 (
           UnitNo                   := #UnitNo,
           ActRec                   := DB2450.RV2_A5,
           Typ                      := 1,
           FBa                      := #xTmp,
           FBa2                     := I    327.6,
           Out                      := Q    327.6);

NETWORK
TITLE =RV3_A5
// Act 007
// Box           : Ventilinsel 3
// Input address : I327.7
// Output address: Q327.7
      CALL FC    70 (
           UnitNo                   := #UnitNo,
           ActRec                   := DB2450.RV3_A5,
           Typ                      := 1,
           FBa                      := #xTmp,
           FBa2                     := I    327.7,
           Out                      := Q    327.7);

NETWORK
TITLE =VR_V1
// Act 008
// Box           : Ventilinsel 4
// Input address : I336.3
// Output address: Q336.3
      CALL FC    70 (
           UnitNo                   := #UnitNo,
           ActRec                   := DB2450.VR_V1,
           Typ                      := 1,
           FBa                      := #xTmp,
           FBa2                     := I    336.3,
           Out                      := Q    336.3);

NETWORK
TITLE =U45_Act010  spare
// Act 010
// Box           :
// Output address: #xtmp
      CALL FC    70 (
           UnitNo                   := #UnitNo,
           ActRec                   := DB2450.U45_Act010,
           Typ                      := 0,
           FBa                      := #xTmp,
           FBa2                     := #xTmp,
           Out                      := #xTmp);

END_FUNCTION_BLOCK

FUNCTION_BLOCK FB 1451
TITLE =U045: Water Transfer Plant 5
FAMILY : BOTEC_F1
NAME : UniE
VERSION : 1.2


VAR_TEMP
  CIP : BOOL ;	//CIP active
  UNIM : BOOL ;	//Unit Not In Maintenance
  GenRel : BOOL ;	//general OK (emergency and maintenance OK)
  EStopOK : BOOL ;	//emergency OK
  UnitNo : INT ;	//unit number
  xTmp : BOOL ;	//Temporary Bool
  iTmp : INT ;	//Temporary INT
  rTmp : REAL ;	//Temporary REAL
  dTmp : DINT ;	//Temporary DINT (free for general use)
  RetValInt : INT ;	//return value
END_VAR
BEGIN
NETWORK
TITLE =General

      SET   ;
// Simulation ---------------------------------------------------------------
      A     DB1451.DBX 1357.7;
      CC    FB  1459; // "U045Sim"
      A     DB1451.DBX   17.3;
      =     DB1451.DBX 1357.7; //Help bit for simulation

// get unit number ----------------------------------------------------------
      L     DB1450.DBW    0;
      T     #UnitNo;

// communication ------------------------------------------------------------
      UC    FB  1455;

NETWORK
TITLE =Sequence organisation

      CLR   ;
      =     M    122.2;

// CIP Counter
      CALL FC    29 (
           UnitNo                   := #UnitNo,
           Value                    := DB1455.DBD   54,
           Enable                   := TRUE,
           Down                     := FALSE,
           OriginDetect             := 0.000000e+000,
           MaxDiffPS                := 1.000000e+000,
           SFMRec                   := DB1451.Seq.SFM[15],
           ValueOld                 := DB1451.DBD 1418);

// sequencer ----------------------------------------------------------------
      A     DB1453.DBX   43.1;
      S     DB1453.DBX   97.3;

      CALL FC    40 (
           UnitNo                   := #UnitNo);

END_FUNCTION_BLOCK

FUNCTION_BLOCK FB 1470
TITLE =U047: Water Transfer Plant 7
FAMILY : BOTEC_F1
NAME : UniA
VERSION : 2.1


VAR_TEMP
  EStopOK : BOOL ;	//auxiliary flag
  CIP : BOOL ;	//CIP Program Selected
  xTmp : BOOL ;	//Temporary Bool(free for general use)
  UnitNo : INT ;	//unit number
  UnitFB : INT ;	//unit expansion FB number
  rTmp : REAL ;	//Temporary REAL (free for general use)
  iTmp : INT ;	//Temporary INT (free for general use)
  dTmp : DINT ;	//Temporary DINT (free for general use)
END_VAR
BEGIN
NETWORK
TITLE =general

      CLR   ;
      =     #xTmp;
      =     #EStopOK;

      L     DB1470.DBW    0;
      T     #UnitNo;
      L     DB1470.DBW    2;
      T     #UnitFB;

NETWORK
TITLE =Universal value

      NOP   0;
// unv001 UnV 001 Process Status
      CALL FC    27 (
           UnitNo                   := #UnitNo,
           UnVRec                   := DB2475.unv001,
           ValExt                   := DB2475.DBD  234);

// unv002 UnV 002 Universal Value 02
      CALL FC    27 (
           UnitNo                   := #UnitNo,
           UnVRec                   := DB2475.unv002,
           ValExt                   := DB2475.DBD  362);

// unv003 UnV 003 Universal Value 03
      CALL FC    27 (
           UnitNo                   := #UnitNo,
           UnVRec                   := DB2475.unv003,
           ValExt                   := DB2475.DBD  490);

// unv004 UnV 004 Universal Value 04
      CALL FC    27 (
           UnitNo                   := #UnitNo,
           UnVRec                   := DB2475.unv004,
           ValExt                   := DB2475.DBD  618);

NETWORK
TITLE =special inputs

      NOP   0;
// U47_SpI001 SpI 001 spare
      CALL FC    14 (
           UnitNo                   := #UnitNo,
           SpIRec                   := DB2471.U47_SpI001,
           SpIBit                   := #xTmp);

NETWORK
TITLE =messages

      NOP   0;
// msg001 Msg 001 Message 01
      CALL FC    16 (
           UnitNo                   := #UnitNo,
           MsgRec                   := DB2477.msg001,
           MsgBit                   := DB2477.DBX   82.7);

// msg002 Msg 002 Message 02
      CALL FC    16 (
           UnitNo                   := #UnitNo,
           MsgRec                   := DB2477.msg002,
           MsgBit                   := DB2477.DBX  142.7);

// msg003 Msg 003 Message 03
      CALL FC    16 (
           UnitNo                   := #UnitNo,
           MsgRec                   := DB2477.msg003,
           MsgBit                   := DB2477.DBX  202.7);

NETWORK
TITLE =unit supply

      UC    FB [#UnitFB];

NETWORK
TITLE =Act1  Wasserpumpe
// Act 001
// Box           :
// Input address : #xTmp
// Output address: #xTmp
      CALL FC    70 (
           UnitNo                   := #UnitNo,
           ActRec                   := DB2470.Act1,
           Typ                      := 0,
           FBa                      := I     59.1,
           FBa2                     := #xTmp,
           Out                      := Q     59.1);

NETWORK
TITLE =A7_V11  Filter Anlage 7
// Act 002
// Box           : VSA7
// Input address : I24.6
// Output address: Q46.6
      CALL FC    70 (
           UnitNo                   := #UnitNo,
           ActRec                   := DB2470.A7_V11,
           Typ                      := 1,
           FBa                      := #xTmp,
           FBa2                     := I     24.6,
           Out                      := Q     46.6);

NETWORK
TITLE =A7_V12  Filter Anlage 7
// Act 003
// Box           : VSA7
// Input address : I24.7
// Output address: Q46.7
      CALL FC    70 (
           UnitNo                   := #UnitNo,
           ActRec                   := DB2470.A7_V12,
           Typ                      := 1,
           FBa                      := #xTmp,
           FBa2                     := I     24.7,
           Out                      := Q     46.7);

NETWORK
TITLE =A7_V13  Filter Anlage 7
// Act 004
// Box           : VSA7
// Input address : I25.0
// Output address: Q47.0
      CALL FC    70 (
           UnitNo                   := #UnitNo,
           ActRec                   := DB2470.A7_V13,
           Typ                      := 1,
           FBa                      := #xTmp,
           FBa2                     := I     25.0,
           Out                      := Q     47.0);

NETWORK
TITLE =RV1_A7
// Act 005
// Box           : Ventilinsel 2
// Input address : I323.5
// Output address: Q323.5
      CALL FC    70 (
           UnitNo                   := #UnitNo,
           ActRec                   := DB2470.RV1_A7,
           Typ                      := 1,
           FBa                      := #xTmp,
           FBa2                     := I    323.5,
           Out                      := Q    323.5);

NETWORK
TITLE =RV2_A7
// Act 006
// Box           : Ventilinsel 2
// Input address : I323.6
// Output address: Q323.6
      CALL FC    70 (
           UnitNo                   := #UnitNo,
           ActRec                   := DB2470.RV2_A7,
           Typ                      := 1,
           FBa                      := #xTmp,
           FBa2                     := I    323.6,
           Out                      := Q    323.6);

NETWORK
TITLE =RV3_A7
// Act 007
// Box           : Ventilinsel 2
// Input address : I323.7
// Output address: Q323.7
      CALL FC    70 (
           UnitNo                   := #UnitNo,
           ActRec                   := DB2470.RV3_A7,
           Typ                      := 1,
           FBa                      := #xTmp,
           FBa2                     := I    323.7,
           Out                      := Q    323.7);

NETWORK
TITLE =VR_V3
// Act 008
// Box           : Ventilinsel 4
// Input address : I336.5
// Output address: Q336.5
      CALL FC    70 (
           UnitNo                   := #UnitNo,
           ActRec                   := DB2470.VR_V3,
           Typ                      := 1,
           FBa                      := #xTmp,
           FBa2                     := I    336.5,
           Out                      := Q    336.5);

NETWORK
TITLE =U47_Act010  spare
// Act 010
// Box           :
// Output address: #xtmp
      CALL FC    70 (
           UnitNo                   := #UnitNo,
           ActRec                   := DB2470.U47_Act010,
           Typ                      := 0,
           FBa                      := #xTmp,
           FBa2                     := #xTmp,
           Out                      := #xTmp);

END_FUNCTION_BLOCK

FUNCTION_BLOCK FB 1471
TITLE =U047: Water Transfer Plant 7
FAMILY : BOTEC_F1
NAME : UniE
VERSION : 1.2


VAR_TEMP
  CIP : BOOL ;	//CIP active
  UNIM : BOOL ;	//Unit Not In Maintenance
  GenRel : BOOL ;	//general OK (emergency and maintenance OK)
  EStopOK : BOOL ;	//emergency OK
  UnitNo : INT ;	//unit number
  xTmp : BOOL ;	//Temporary Bool
  iTmp : INT ;	//Temporary INT
  rTmp : REAL ;	//Temporary REAL
  dTmp : DINT ;	//Temporary DINT (free for general use)
  RetValInt : INT ;	//return value
END_VAR
BEGIN
NETWORK
TITLE =General

      SET   ;
// Simulation ---------------------------------------------------------------
      A     DB1471.DBX 1357.7;
      CC    FB  1479; // "U047Sim"
      A     DB1471.DBX   17.3;
      =     DB1471.DBX 1357.7; //Help bit for simulation

// get unit number ----------------------------------------------------------
      L     DB1470.DBW    0;
      T     #UnitNo;

// communication ------------------------------------------------------------
      UC    FB  1475;

NETWORK
TITLE =Sequence organisation

      CLR   ;
      =     M    122.2;

// CIP Counter
      CALL FC    29 (
           UnitNo                   := #UnitNo,
           Value                    := DB1475.DBD   54,
           Enable                   := TRUE,
           Down                     := FALSE,
           OriginDetect             := 0.000000e+000,
           MaxDiffPS                := 1.000000e+000,
           SFMRec                   := DB1471.Seq.SFM[15],
           ValueOld                 := DB1471.DBD 1418);

// sequencer ----------------------------------------------------------------
      A     DB1473.DBX   43.1;
      S     DB1473.DBX   97.3;

      CALL FC    40 (
           UnitNo                   := #UnitNo);

END_FUNCTION_BLOCK

FUNCTION_BLOCK FB 1480
TITLE =U048: Water Transfer Plant 8
FAMILY : BOTEC_F1
NAME : UniA
VERSION : 2.1


VAR_TEMP
  EStopOK : BOOL ;	//auxiliary flag
  CIP : BOOL ;	//CIP Program Selected
  xTmp : BOOL ;	//Temporary Bool(free for general use)
  UnitNo : INT ;	//unit number
  UnitFB : INT ;	//unit expansion FB number
  rTmp : REAL ;	//Temporary REAL (free for general use)
  iTmp : INT ;	//Temporary INT (free for general use)
  dTmp : DINT ;	//Temporary DINT (free for general use)
END_VAR
BEGIN
NETWORK
TITLE =general

      CLR   ;
      =     #xTmp;
      =     #EStopOK;

      L     DB1480.DBW    0;
      T     #UnitNo;
      L     DB1480.DBW    2;
      T     #UnitFB;

NETWORK
TITLE =Universal value

      NOP   0;
// unv001 UnV 001 Process Status
      CALL FC    27 (
           UnitNo                   := #UnitNo,
           UnVRec                   := DB2485.unv001,
           ValExt                   := DB2485.DBD  234);

// unv002 UnV 002 Universal Value 02
      CALL FC    27 (
           UnitNo                   := #UnitNo,
           UnVRec                   := DB2485.unv002,
           ValExt                   := DB2485.DBD  362);

// unv003 UnV 003 Universal Value 03
      CALL FC    27 (
           UnitNo                   := #UnitNo,
           UnVRec                   := DB2485.unv003,
           ValExt                   := DB2485.DBD  490);

// unv004 UnV 004 Universal Value 04
      CALL FC    27 (
           UnitNo                   := #UnitNo,
           UnVRec                   := DB2485.unv004,
           ValExt                   := DB2485.DBD  618);

NETWORK
TITLE =special inputs

      NOP   0;
// U48_SpI001 SpI 001 spare
      CALL FC    14 (
           UnitNo                   := #UnitNo,
           SpIRec                   := DB2481.U48_SpI001,
           SpIBit                   := #xTmp);

NETWORK
TITLE =messages

      NOP   0;
// msg001 Msg 001 Message 01
      CALL FC    16 (
           UnitNo                   := #UnitNo,
           MsgRec                   := DB2487.msg001,
           MsgBit                   := DB2487.DBX   82.7);

// msg002 Msg 002 Message 02
      CALL FC    16 (
           UnitNo                   := #UnitNo,
           MsgRec                   := DB2487.msg002,
           MsgBit                   := DB2487.DBX  142.7);

// msg003 Msg 003 Message 03
      CALL FC    16 (
           UnitNo                   := #UnitNo,
           MsgRec                   := DB2487.msg003,
           MsgBit                   := DB2487.DBX  202.7);

NETWORK
TITLE =unit supply

      UC    FB [#UnitFB];

NETWORK
TITLE =Pumpe
// Act 005
// Box           : Ventilinsel 3
// Input address : I325.5
// Output address: Q325.5
      CALL FC    70 (
           UnitNo                   := #UnitNo,
           ActRec                   := DB2480.Act1,
           Typ                      := 0,
           FBa                      := #xTmp,
           FBa2                     := #xTmp,
           Out                      := #xTmp);

NETWORK
TITLE =RV1_A8
// Act 005
// Box           : Ventilinsel 3
// Input address : I325.5
// Output address: Q325.5
      CALL FC    70 (
           UnitNo                   := #UnitNo,
           ActRec                   := DB2480.RV1_A8,
           Typ                      := 1,
           FBa                      := #xTmp,
           FBa2                     := I    325.5,
           Out                      := Q    325.5);

NETWORK
TITLE =RV2_A8
// Act 006
// Box           : Ventilinsel 3
// Input address : I325.6
// Output address: Q325.6
      CALL FC    70 (
           UnitNo                   := #UnitNo,
           ActRec                   := DB2480.RV2_A8,
           Typ                      := 1,
           FBa                      := #xTmp,
           FBa2                     := I    325.6,
           Out                      := Q    325.6);

NETWORK
TITLE =RV3_A8
// Act 007
// Box           : Ventilinsel 3
// Input address : I325.7
// Output address: Q325.7
      CALL FC    70 (
           UnitNo                   := #UnitNo,
           ActRec                   := DB2480.RV3_A8,
           Typ                      := 1,
           FBa                      := #xTmp,
           FBa2                     := I    325.7,
           Out                      := Q    325.7);

NETWORK
TITLE =VR_V2
// Act 008
// Box           : Ventilinsel 4
// Input address : I336.4
// Output address: Q336.4
      CALL FC    70 (
           UnitNo                   := #UnitNo,
           ActRec                   := DB2480.VR_V2,
           Typ                      := 1,
           FBa                      := #xTmp,
           FBa2                     := I    336.4,
           Out                      := Q    336.4);

NETWORK
TITLE =U48_Act010  spare
// Act 010
// Box           :
// Output address: #xtmp
      CALL FC    70 (
           UnitNo                   := #UnitNo,
           ActRec                   := DB2480.U48_Act010,
           Typ                      := 0,
           FBa                      := #xTmp,
           FBa2                     := #xTmp,
           Out                      := #xTmp);

END_FUNCTION_BLOCK

FUNCTION_BLOCK FB 1481
TITLE =U048: Water Transfer Plant 8
FAMILY : BOTEC_F1
NAME : UniE
VERSION : 1.2


VAR_TEMP
  CIP : BOOL ;	//CIP active
  UNIM : BOOL ;	//Unit Not In Maintenance
  GenRel : BOOL ;	//general OK (emergency and maintenance OK)
  EStopOK : BOOL ;	//emergency OK
  UnitNo : INT ;	//unit number
  xTmp : BOOL ;	//Temporary Bool
  iTmp : INT ;	//Temporary INT
  rTmp : REAL ;	//Temporary REAL
  dTmp : DINT ;	//Temporary DINT (free for general use)
  RetValInt : INT ;	//return value
END_VAR
BEGIN
NETWORK
TITLE =General

      SET   ;
// Simulation ---------------------------------------------------------------
      A     DB1481.DBX 1357.7;
      CC    FB  1489; // "U048Sim"
      A     DB1481.DBX   17.3;
      =     DB1481.DBX 1357.7; //Help bit for simulation

// get unit number ----------------------------------------------------------
      L     DB1480.DBW    0;
      T     #UnitNo;

// communication ------------------------------------------------------------
      UC    FB  1485; // U048Com

NETWORK
TITLE =Sequence organisation

      CLR   ;
      =     M    122.2;

// sequencer ----------------------------------------------------------------
      A     DB1483.DBX   43.1;
      S     DB1483.DBX   97.3;

      CALL FC    40 (
           UnitNo                   := #UnitNo);

END_FUNCTION_BLOCK

FUNCTION_BLOCK FB 1490
TITLE =U049: Water Transfer Plant 9
FAMILY : BOTEC_F1
NAME : UniA
VERSION : 2.1


VAR_TEMP
  EStopOK : BOOL ;	//auxiliary flag
  CIP : BOOL ;	//CIP Program Selected
  xTmp : BOOL ;	//Temporary Bool(free for general use)
  UnitNo : INT ;	//unit number
  UnitFB : INT ;	//unit expansion FB number
  rTmp : REAL ;	//Temporary REAL (free for general use)
  iTmp : INT ;	//Temporary INT (free for general use)
  dTmp : DINT ;	//Temporary DINT (free for general use)
END_VAR
BEGIN
NETWORK
TITLE =general

      CLR   ;
      =     #xTmp;
      =     #EStopOK;

      L     DB1490.DBW    0;
      T     #UnitNo;
      L     DB1490.DBW    2;
      T     #UnitFB;

NETWORK
TITLE =Universal value

      NOP   0;
// unv001 UnV 001 Process Status
      CALL FC    27 (
           UnitNo                   := #UnitNo,
           UnVRec                   := DB2495.unv001,
           ValExt                   := DB2495.DBD  234);

// unv002 UnV 002 Universal Value 02
      CALL FC    27 (
           UnitNo                   := #UnitNo,
           UnVRec                   := DB2495.unv002,
           ValExt                   := DB2495.DBD  362);

// unv003 UnV 003 Universal Value 03
      CALL FC    27 (
           UnitNo                   := #UnitNo,
           UnVRec                   := DB2495.unv003,
           ValExt                   := DB2495.DBD  490);

// unv004 UnV 004 Universal Value 04
      CALL FC    27 (
           UnitNo                   := #UnitNo,
           UnVRec                   := DB2495.unv004,
           ValExt                   := DB2495.DBD  618);

NETWORK
TITLE =special inputs

      NOP   0;
// U49_SpI001 SpI 001 spare
      CALL FC    14 (
           UnitNo                   := #UnitNo,
           SpIRec                   := DB2491.U49_SpI001,
           SpIBit                   := #xTmp);

NETWORK
TITLE =messages

      NOP   0;
// msg001 Msg 001 Message 01
      CALL FC    16 (
           UnitNo                   := #UnitNo,
           MsgRec                   := DB2497.msg001,
           MsgBit                   := DB2497.DBX   82.7);

// msg002 Msg 002 Message 02
      CALL FC    16 (
           UnitNo                   := #UnitNo,
           MsgRec                   := DB2497.msg002,
           MsgBit                   := DB2497.DBX  142.7);

// msg003 Msg 003 Message 03
      CALL FC    16 (
           UnitNo                   := #UnitNo,
           MsgRec                   := DB2497.msg003,
           MsgBit                   := DB2497.DBX  202.7);

NETWORK
TITLE =unit supply

      UC    FB [#UnitFB];

NETWORK
TITLE =Act1  Wasserpumpe
// Act 001
// Box           :
// Input address : #xTmp
// Output address: #xTmp
      CALL FC    70 (
           UnitNo                   := #UnitNo,
           ActRec                   := DB2490.Act1,
           Typ                      := 0,
           FBa                      := #xTmp,
           FBa2                     := #xTmp,
           Out                      := Q     41.1);

NETWORK
TITLE =A9_V11  Ventil Filter Anlage 9
// Act 002
// Box           : VSRR1-3
// Input address : I85.4
// Output address: Q85.4
      CALL FC    70 (
           UnitNo                   := #UnitNo,
           ActRec                   := DB2490.A9_V11,
           Typ                      := 1,
           FBa                      := #xTmp,
           FBa2                     := I     85.4,
           Out                      := Q     85.4);

NETWORK
TITLE =A9_V12  Ventil Filter Anlage 9
// Act 003
// Box           : VSRR1-3
// Input address : I85.5
// Output address: Q85.5
      CALL FC    70 (
           UnitNo                   := #UnitNo,
           ActRec                   := DB2490.A9_V12,
           Typ                      := 1,
           FBa                      := #xTmp,
           FBa2                     := I     85.5,
           Out                      := Q     85.5);

NETWORK
TITLE =A9_V13  Ventil Filter Anlage 9
// Act 004
// Box           : VSRR1-3
// Input address : I85.6
// Output address: Q85.6
      CALL FC    70 (
           UnitNo                   := #UnitNo,
           ActRec                   := DB2490.A9_V13,
           Typ                      := 1,
           FBa                      := #xTmp,
           FBa2                     := I     85.6,
           Out                      := Q     85.6);

NETWORK
TITLE =RV1_A9
// Act 005
// Box           : Ventilinsel 2
// Input address : I319.5
// Output address: Q319.5
      CALL FC    70 (
           UnitNo                   := #UnitNo,
           ActRec                   := DB2490.RV1_A9,
           Typ                      := 1,
           FBa                      := #xTmp,
           FBa2                     := I    319.5,
           Out                      := Q    319.5);

NETWORK
TITLE =RV2_A9
// Act 006
// Box           : Ventilinsel 2
// Input address : I319.6
// Output address: Q319.6
      CALL FC    70 (
           UnitNo                   := #UnitNo,
           ActRec                   := DB2490.RV2_A9,
           Typ                      := 1,
           FBa                      := #xTmp,
           FBa2                     := I    319.6,
           Out                      := Q    319.6);

NETWORK
TITLE =RV3_A9
// Act 007
// Box           : Ventilinsel 2
// Input address : I319.7
// Output address: Q319.7
      CALL FC    70 (
           UnitNo                   := #UnitNo,
           ActRec                   := DB2490.RV3_A9,
           Typ                      := 1,
           FBa                      := #xTmp,
           FBa2                     := I    319.7,
           Out                      := Q    319.7);

NETWORK
TITLE =VR_V5
// Act 008
// Box           : Ventilinsel 4
// Input address : I336.7
// Output address: Q336.7
      CALL FC    70 (
           UnitNo                   := #UnitNo,
           ActRec                   := DB2490.VR_V5,
           Typ                      := 1,
           FBa                      := #xTmp,
           FBa2                     := I    336.7,
           Out                      := Q    336.7);

NETWORK
TITLE =U49_Act010  spare
// Act 010
// Box           :
// Output address: #xtmp
      CALL FC    70 (
           UnitNo                   := #UnitNo,
           ActRec                   := DB2490.U49_Act010,
           Typ                      := 0,
           FBa                      := #xTmp,
           FBa2                     := #xTmp,
           Out                      := #xTmp);

END_FUNCTION_BLOCK

FUNCTION_BLOCK FB 1491
TITLE =U049: Water Transfer Plant 9
FAMILY : BOTEC_F1
NAME : UniE
VERSION : 1.2


VAR_TEMP
  CIP : BOOL ;	//CIP active
  UNIM : BOOL ;	//Unit Not In Maintenance
  GenRel : BOOL ;	//general OK (emergency and maintenance OK)
  EStopOK : BOOL ;	//emergency OK
  UnitNo : INT ;	//unit number
  xTmp : BOOL ;	//Temporary Bool
  iTmp : INT ;	//Temporary INT
  rTmp : REAL ;	//Temporary REAL
  dTmp : DINT ;	//Temporary DINT (free for general use)
  RetValInt : INT ;	//return value
END_VAR
BEGIN
NETWORK
TITLE =General

      SET   ;
// Simulation ---------------------------------------------------------------
      A     DB1491.DBX 1357.7;
      CC    FB  1499; // "U049Sim"
      A     DB1491.DBX   17.3;
      =     DB1491.DBX 1357.7; //Help bit for simulation

// get unit number ----------------------------------------------------------
      L     DB1490.DBW    0;
      T     #UnitNo;

// communication ------------------------------------------------------------
      UC    FB  1495;

NETWORK
TITLE =Sequence organisation

      CLR   ;
      =     M    122.2;

// CIP Counter
      CALL FC    29 (
           UnitNo                   := #UnitNo,
           Value                    := DB1495.DBD   54,
           Enable                   := TRUE,
           Down                     := FALSE,
           OriginDetect             := 0.000000e+000,
           MaxDiffPS                := 1.000000e+000,
           SFMRec                   := DB1491.Seq.SFM[15],
           ValueOld                 := DB1491.DBD 1418);

// sequencer ----------------------------------------------------------------
      A     DB1493.DBX   43.1;
      S     DB1493.DBX   97.3;

      CALL FC    40 (
           UnitNo                   := #UnitNo);

END_FUNCTION_BLOCK

FUNCTION_BLOCK FB 1500
TITLE =U050: Water Transfer Plant 10
FAMILY : BOTEC_F1
NAME : UniA
VERSION : 2.1


VAR_TEMP
  EStopOK : BOOL ;	//auxiliary flag
  CIP : BOOL ;	//CIP Program Selected
  xTmp : BOOL ;	//Temporary Bool(free for general use)
  UnitNo : INT ;	//unit number
  UnitFB : INT ;	//unit expansion FB number
  rTmp : REAL ;	//Temporary REAL (free for general use)
  iTmp : INT ;	//Temporary INT (free for general use)
  dTmp : DINT ;	//Temporary DINT (free for general use)
END_VAR
BEGIN
NETWORK
TITLE =general

      CLR   ;
      =     #xTmp;
      =     #EStopOK;

      L     DB1500.DBW    0;
      T     #UnitNo;
      L     DB1500.DBW    2;
      T     #UnitFB;

NETWORK
TITLE =Universal value

      NOP   0;
// unv001 UnV 001 Process Status
      CALL FC    27 (
           UnitNo                   := #UnitNo,
           UnVRec                   := DB2505.unv001,
           ValExt                   := DB2505.DBD  234);

// unv002 UnV 002 Universal Value 02
      CALL FC    27 (
           UnitNo                   := #UnitNo,
           UnVRec                   := DB2505.unv002,
           ValExt                   := DB2505.DBD  362);

// unv003 UnV 003 Universal Value 03
      CALL FC    27 (
           UnitNo                   := #UnitNo,
           UnVRec                   := DB2505.unv003,
           ValExt                   := DB2505.DBD  490);

// unv004 UnV 004 Universal Value 04
      CALL FC    27 (
           UnitNo                   := #UnitNo,
           UnVRec                   := DB2505.unv004,
           ValExt                   := DB2505.DBD  618);

NETWORK
TITLE =special inputs

      NOP   0;
// U50_SpI001 SpI 001 spare
      CALL FC    14 (
           UnitNo                   := #UnitNo,
           SpIRec                   := DB2501.U50_SpI001,
           SpIBit                   := #xTmp);

NETWORK
TITLE =messages

      NOP   0;
// msg001 Msg 001 Message 01
      CALL FC    16 (
           UnitNo                   := #UnitNo,
           MsgRec                   := DB2507.msg001,
           MsgBit                   := DB2507.DBX   82.7);

// msg002 Msg 002 Message 02
      CALL FC    16 (
           UnitNo                   := #UnitNo,
           MsgRec                   := DB2507.msg002,
           MsgBit                   := DB2507.DBX  142.7);

// msg003 Msg 003 Message 03
      CALL FC    16 (
           UnitNo                   := #UnitNo,
           MsgRec                   := DB2507.msg003,
           MsgBit                   := DB2507.DBX  202.7);

NETWORK
TITLE =unit supply

      UC    FB [#UnitFB];

NETWORK
TITLE =Act1  Wasserpumpe
// Act 001
// Box           :
// Input address : #xTmp
// Output address: #xTmp
      CALL FC    70 (
           UnitNo                   := #UnitNo,
           ActRec                   := DB2500.Act1,
           Typ                      := 0,
           FBa                      := I     41.5,
           FBa2                     := #xTmp,
           Out                      := Q     41.5);

NETWORK
TITLE =A10_V11  Ventil Filter Anlage 10
// Act 002
// Box           : VSRR1-3
// Input address : I85.1
// Output address: Q85.1
      CALL FC    70 (
           UnitNo                   := #UnitNo,
           ActRec                   := DB2500.A10_V11,
           Typ                      := 1,
           FBa                      := #xTmp,
           FBa2                     := I     85.1,
           Out                      := Q     85.1);

NETWORK
TITLE =A10_V12  Ventil Filter Anlage 10
// Act 003
// Box           : VSRR1-3
// Input address : I85.2
// Output address: Q85.2
      CALL FC    70 (
           UnitNo                   := #UnitNo,
           ActRec                   := DB2500.A10_V12,
           Typ                      := 1,
           FBa                      := #xTmp,
           FBa2                     := I     85.2,
           Out                      := Q     85.2);

NETWORK
TITLE =A10_V13  Ventil Filter Anlage 10
// Act 004
// Box           : VSRR1-3
// Input address : I85.3
// Output address: Q85.3
      CALL FC    70 (
           UnitNo                   := #UnitNo,
           ActRec                   := DB2500.A10_V13,
           Typ                      := 1,
           FBa                      := #xTmp,
           FBa2                     := I     85.3,
           Out                      := Q     85.3);

NETWORK
TITLE =RV1_A10
// Act 005
// Box           : Ventilinsel 2
// Input address : I317.5
// Output address: Q317.5
      CALL FC    70 (
           UnitNo                   := #UnitNo,
           ActRec                   := DB2500.RV1_A10,
           Typ                      := 1,
           FBa                      := #xTmp,
           FBa2                     := I    317.5,
           Out                      := Q    317.5);

NETWORK
TITLE =RV2_A10
// Act 006
// Box           : Ventilinsel 2
// Input address : I317.6
// Output address: Q317.6
      CALL FC    70 (
           UnitNo                   := #UnitNo,
           ActRec                   := DB2500.RV2_A10,
           Typ                      := 1,
           FBa                      := #xTmp,
           FBa2                     := I    317.6,
           Out                      := Q    317.6);

NETWORK
TITLE =RV3_A10
// Act 007
// Box           : Ventilinsel 2
// Input address : I317.7
// Output address: Q317.7
      CALL FC    70 (
           UnitNo                   := #UnitNo,
           ActRec                   := DB2500.RV3_A10,
           Typ                      := 1,
           FBa                      := #xTmp,
           FBa2                     := I    317.7,
           Out                      := Q    317.7);

NETWORK
TITLE =VR_V6
// Act 008
// Box           : Ventilinsel 4
// Input address : I337.0
// Output address: Q337.0
      CALL FC    70 (
           UnitNo                   := #UnitNo,
           ActRec                   := DB2500.VR_V6,
           Typ                      := 1,
           FBa                      := #xTmp,
           FBa2                     := I    337.0,
           Out                      := Q    337.0);

NETWORK
TITLE =U50_Act010  spare
// Act 010
// Box           :
// Output address: #xtmp
      CALL FC    70 (
           UnitNo                   := #UnitNo,
           ActRec                   := DB2500.U50_Act010,
           Typ                      := 0,
           FBa                      := #xTmp,
           FBa2                     := #xTmp,
           Out                      := #xTmp);

END_FUNCTION_BLOCK

FUNCTION_BLOCK FB 1501
TITLE =U050: Water Transfer Plant 10
FAMILY : BOTEC_F1
NAME : UniE
VERSION : 1.2


VAR_TEMP
  CIP : BOOL ;	//CIP active
  UNIM : BOOL ;	//Unit Not In Maintenance
  GenRel : BOOL ;	//general OK (emergency and maintenance OK)
  EStopOK : BOOL ;	//emergency OK
  UnitNo : INT ;	//unit number
  xTmp : BOOL ;	//Temporary Bool
  iTmp : INT ;	//Temporary INT
  rTmp : REAL ;	//Temporary REAL
  dTmp : DINT ;	//Temporary DINT (free for general use)
  RetValInt : INT ;	//return value
END_VAR
BEGIN
NETWORK
TITLE =General

      SET   ;
// Simulation ---------------------------------------------------------------
      A     DB1501.DBX 1357.7;
      CC    FB  1509; // "U050Sim"
      A     DB1501.DBX   17.3;
      =     DB1501.DBX 1357.7; //Help bit for simulation

// get unit number ----------------------------------------------------------
      L     DB1500.DBW    0;
      T     #UnitNo;

// communication ------------------------------------------------------------
      UC    FB  1505; // U050Com

NETWORK
TITLE =Sequence organisation

      CLR   ;
      =     M    122.2;

// CIP Counter
      CALL FC    29 (
           UnitNo                   := #UnitNo,
           Value                    := DB1505.DBD   54,
           Enable                   := TRUE,
           Down                     := FALSE,
           OriginDetect             := 0.000000e+000,
           MaxDiffPS                := 1.000000e+000,
           SFMRec                   := DB1501.Seq.SFM[15],
           ValueOld                 := DB1501.DBD 1418);

// sequencer ----------------------------------------------------------------
      A     DB1503.DBX   43.1;
      S     DB1503.DBX   97.3;

      CALL FC    40 (
           UnitNo                   := #UnitNo);

END_FUNCTION_BLOCK

FUNCTION_BLOCK FB 1510
TITLE =U051: Water Transfer Plant 11
FAMILY : BOTEC_F1
NAME : UniA
VERSION : 2.1


VAR_TEMP
  EStopOK : BOOL ;	//auxiliary flag
  CIP : BOOL ;	//CIP Program Selected
  xTmp : BOOL ;	//Temporary Bool(free for general use)
  UnitNo : INT ;	//unit number
  UnitFB : INT ;	//unit expansion FB number
  rTmp : REAL ;	//Temporary REAL (free for general use)
  iTmp : INT ;	//Temporary INT (free for general use)
  dTmp : DINT ;	//Temporary DINT (free for general use)
END_VAR
BEGIN
NETWORK
TITLE =general

      CLR   ;
      =     #xTmp;
      =     #EStopOK;

      L     DB1510.DBW    0;
      T     #UnitNo;
      L     DB1510.DBW    2;
      T     #UnitFB;

NETWORK
TITLE =Universal value

      NOP   0;
// unv001 UnV 001 Process Status
      CALL FC    27 (
           UnitNo                   := #UnitNo,
           UnVRec                   := DB2515.unv001,
           ValExt                   := DB2515.DBD  234);

// unv002 UnV 002 Universal Value 02
      CALL FC    27 (
           UnitNo                   := #UnitNo,
           UnVRec                   := DB2515.unv002,
           ValExt                   := DB2515.DBD  362);

// unv003 UnV 003 Universal Value 03
      CALL FC    27 (
           UnitNo                   := #UnitNo,
           UnVRec                   := DB2515.unv003,
           ValExt                   := DB2515.DBD  490);

// unv004 UnV 004 Universal Value 04
      CALL FC    27 (
           UnitNo                   := #UnitNo,
           UnVRec                   := DB2515.unv004,
           ValExt                   := DB2515.DBD  618);

NETWORK
TITLE =special inputs

      NOP   0;
// U51_SpI001 SpI 001 spare
      CALL FC    14 (
           UnitNo                   := #UnitNo,
           SpIRec                   := DB2511.U51_SpI001,
           SpIBit                   := #xTmp);

NETWORK
TITLE =messages

      NOP   0;
// msg001 Msg 001 Message 01
      CALL FC    16 (
           UnitNo                   := #UnitNo,
           MsgRec                   := DB2517.msg001,
           MsgBit                   := DB2517.DBX   82.7);

// msg002 Msg 002 Message 02
      CALL FC    16 (
           UnitNo                   := #UnitNo,
           MsgRec                   := DB2517.msg002,
           MsgBit                   := DB2517.DBX  142.7);

// msg003 Msg 003 Message 03
      CALL FC    16 (
           UnitNo                   := #UnitNo,
           MsgRec                   := DB2517.msg003,
           MsgBit                   := DB2517.DBX  202.7);

NETWORK
TITLE =unit supply

      UC    FB [#UnitFB];

NETWORK
TITLE =Act1  Wasserpumpe
// Act 001
// Box           :
// Input address : #xTmp
// Output address: #xTmp
      CALL FC    70 (
           UnitNo                   := #UnitNo,
           ActRec                   := DB2510.Act1,
           Typ                      := 0,
           FBa                      := I    171.1,
           FBa2                     := #xTmp,
           Out                      := Q    171.1);

NETWORK
TITLE =A11_V11  A11 V11
// Act 002
// Box           : VSA11
// Input address : I174.6
// Output address: Q174.6
      CALL FC    70 (
           UnitNo                   := #UnitNo,
           ActRec                   := DB2510.A11_V11,
           Typ                      := 1,
           FBa                      := #xTmp,
           FBa2                     := I    174.6,
           Out                      := Q    174.6);

NETWORK
TITLE =A11_V12  A11 V12
// Act 003
// Box           : VSA11
// Input address : I174.7
// Output address: Q174.7
      CALL FC    70 (
           UnitNo                   := #UnitNo,
           ActRec                   := DB2510.A11_V12,
           Typ                      := 1,
           FBa                      := #xTmp,
           FBa2                     := I    174.7,
           Out                      := Q    174.7);

NETWORK
TITLE =A11_V13  A11 V13
// Act 004
// Box           : VSA11
// Input address : I175.0
// Output address: Q175.0
      CALL FC    70 (
           UnitNo                   := #UnitNo,
           ActRec                   := DB2510.A11_V13,
           Typ                      := 1,
           FBa                      := #xTmp,
           FBa2                     := I    175.0,
           Out                      := Q    175.0);

NETWORK
TITLE =RV1_A11
// Act 005
// Box           : Ventilinsel 3
// Input address : I329.5
// Output address: Q329.5
      CALL FC    70 (
           UnitNo                   := #UnitNo,
           ActRec                   := DB2510.RV1_A11,
           Typ                      := 1,
           FBa                      := #xTmp,
           FBa2                     := I    329.5,
           Out                      := Q    329.5);

NETWORK
TITLE =RV2_A11
// Act 006
// Box           : Ventilinsel 3
// Input address : I329.6
// Output address: Q329.6
      CALL FC    70 (
           UnitNo                   := #UnitNo,
           ActRec                   := DB2510.RV2_A11,
           Typ                      := 1,
           FBa                      := #xTmp,
           FBa2                     := I    329.6,
           Out                      := Q    329.6);

NETWORK
TITLE =RV3_A11
// Act 007
// Box           : Ventilinsel 3
// Input address : I329.7
// Output address: Q329.7
      CALL FC    70 (
           UnitNo                   := #UnitNo,
           ActRec                   := DB2510.RV3_A11,
           Typ                      := 1,
           FBa                      := #xTmp,
           FBa2                     := I    329.7,
           Out                      := Q    329.7);

NETWORK
TITLE =VR_V10
// Act 008
// Box           : Ventilinsel 4
// Input address : I336.2
// Output address: Q336.2
      CALL FC    70 (
           UnitNo                   := #UnitNo,
           ActRec                   := DB2510.VR_V10,
           Typ                      := 1,
           FBa                      := #xTmp,
           FBa2                     := I    336.2,
           Out                      := Q    336.2);

NETWORK
TITLE =VR_V7
// Act 009
// Box           : Ventilinsel 4
// Input address : I337.1
// Output address: Q337.1
      CALL FC    70 (
           UnitNo                   := #UnitNo,
           ActRec                   := DB2510.VR_V7,
           Typ                      := 1,
           FBa                      := #xTmp,
           FBa2                     := I    337.1,
           Out                      := Q    337.1);

NETWORK
TITLE =U51_Act010  spare
// Act 010
// Box           :
// Output address: #xtmp
      CALL FC    70 (
           UnitNo                   := #UnitNo,
           ActRec                   := DB2510.U51_Act010,
           Typ                      := 0,
           FBa                      := #xTmp,
           FBa2                     := #xTmp,
           Out                      := #xTmp);

END_FUNCTION_BLOCK

FUNCTION_BLOCK FB 1511
TITLE =U051: Water Transfer Plant 11
FAMILY : BOTEC_F1
NAME : UniE
VERSION : 1.2


